stPrcRecipe.stUBL.nRecipeIndexShow.diValue															:=		stPrcRecipe.stUBL.nRecipeIndexShow.diDefault															 ;
stPrcRecipe.stUBL.iPackageCapTypeShow.diValue														:=      stPrcRecipe.stUBL.iPackageCapTypeShow.diDefault														     ;
stPrcRecipe.stUBL.iPackageCapDiameterShow.diValue 													:=      stPrcRecipe.stUBL.iPackageCapDiameterShow.diDefault 													 ;
stPrcRecipe.stUBL.bExEnableShow.bValue 																:=      stPrcRecipe.stUBL.bExEnableShow.bDefault															     ;
stPrcRecipe.stUBL.bBottleFeederEnableShow.bValue													:=      stPrcRecipe.stUBL.bBottleFeederEnableShow.bDefault													     ;
stPrcRecipe.stUBL.iBottleFeederTurntableVelocitySVShow.udiValue										:=      stPrcRecipe.stUBL.iBottleFeederTurntableVelocitySVShow.udiDefault										 ;
stPrcRecipe.stUBL.iBottleFeederBottleSensorDelayShow.diValue										:=      stPrcRecipe.stUBL.iBottleFeederBottleSensorDelayShow.diDefault										     ;
stPrcRecipe.stUBL.iBottleFeederFormGateDelayShow.diValue											:=      stPrcRecipe.stUBL.iBottleFeederFormGateDelayShow.diDefault											     ;
stPrcRecipe.stUBL.iBottleFeederAllowFormDelayShow.diValue											:=      stPrcRecipe.stUBL.iBottleFeederAllowFormDelayShow.diDefault											     ;
stPrcRecipe.stUBL.bPucksInserterEnableShow.bValue													:=      stPrcRecipe.stUBL.bPucksInserterEnableShow.bDefault												         ;
stPrcRecipe.stUBL.iPucksInserterTurntableVelocitySVShow.udiValue 									:=      stPrcRecipe.stUBL.iPucksInserterTurntableVelocitySVShow.udiDefault									     ;
stPrcRecipe.stUBL.iPucksInserterConveyorVelocitySVShow.udiValue										:=      stPrcRecipe.stUBL.iPucksInserterConveyorVelocitySVShow.udiDefault									     ;
stPrcRecipe.stUBL.iPucksInserterBottleSensorDelayShow.diValue										:=      stPrcRecipe.stUBL.iPucksInserterBottleSensorDelayShow.diDefault										     ;
stPrcRecipe.stUBL.iPucksInserterFormGateDelayShow.diValue 											:=      stPrcRecipe.stUBL.iPucksInserterFormGateDelayShow.diDefault 											 ;
stPrcRecipe.stUBL.iPucksInserterAllowFormDelayShow.diValue 											:=      stPrcRecipe.stUBL.iPucksInserterAllowFormDelayShow.diDefault											 ;
stPrcRecipe.stUBL.lrPucksInserterWheelOffsetShow.lrValue 											:=      stPrcRecipe.stUBL.lrPucksInserterWheelOffsetShow.lrDefault											     ;
stPrcRecipe.stUBL.lrPucksInserterWheelAccelerationShow.lrValue 										:=      stPrcRecipe.stUBL.lrPucksInserterWheelAccelerationShow.lrDefault										 ;
stPrcRecipe.stUBL.lrPucksInserterWheelVelocityShow.lrValue 											:=      stPrcRecipe.stUBL.lrPucksInserterWheelVelocityShow.lrDefault											 ;
stPrcRecipe.stUBL.lrPucksInserterHammerHeightSVShow.lrValue 										:=      stPrcRecipe.stUBL.lrPucksInserterHammerHeightSVShow.lrDefault	 										 ;
stPrcRecipe.stUBL.bGateBeforeDispencersEnableShow.bValue											:=      stPrcRecipe.stUBL.bGateBeforeDispencersEnableShow.bDefault									             ;
stPrcRecipe.stUBL.nGateBeforeDispencersTimeFormInsertingShow.lrValue 								:=      stPrcRecipe.stUBL.nGateBeforeDispencersTimeFormInsertingShow.lrDefault								     ;
stPrcRecipe.stUBL.bGateAfterWeightEnableShow.bValue 												:=      stPrcRecipe.stUBL.bGateAfterWeightEnableShow.bDefault												     ;
stPrcRecipe.stUBL.nGateAfterWeightTimeFormInsertingShow.lrValue 									:=      stPrcRecipe.stUBL.nGateAfterWeightTimeFormInsertingShow.lrDefault									     ;
stPrcRecipe.stUBL.bGateRobotEnableShow.bValue       												:=      stPrcRecipe.stUBL.bGateRobotEnableShow.bDefault    												         ;
stPrcRecipe.stUBL.nGateRobotTimeFormInsertingShow.lrValue											:=      stPrcRecipe.stUBL.nGateRobotTimeFormInsertingShow.lrDefault											     ;
stPrcRecipe.stUBL.bFormsDragingLeftEnableShow.bValue         										:=      stPrcRecipe.stUBL.bFormsDragingLeftEnableShow.bDefault       										     ;
stPrcRecipe.stUBL.lrFormsDragingLeftVelocityShow.lrValue         									:=      stPrcRecipe.stUBL.lrFormsDragingLeftVelocityShow.lrDefault	     									     ;
stPrcRecipe.stUBL.lrFormsDragingLeftAccelerationShow.lrValue 										:=      stPrcRecipe.stUBL.lrFormsDragingLeftAccelerationShow.lrDefault											 ;
stPrcRecipe.stUBL.lrFormsDragingLeftDecelerationShow.lrValue   										:=      stPrcRecipe.stUBL.lrFormsDragingLeftDecelerationShow.lrDefault											 ;
stPrcRecipe.stUBL.bFormsDragingRightEnableShow.bValue 												:=      stPrcRecipe.stUBL.bFormsDragingRightEnableShow.bDefault											         ;
stPrcRecipe.stUBL.lrFormsDragingRightVelocityShow.lrValue 											:=      stPrcRecipe.stUBL.lrFormsDragingRightVelocityShow.lrDefault												 ;
stPrcRecipe.stUBL.lrFormsDragingRightAccelerationShow.lrValue 										:=      stPrcRecipe.stUBL.lrFormsDragingRightAccelerationShow.lrDefault											 ;
stPrcRecipe.stUBL.lrFormsDragingRightDecelerationShow.lrValue 										:=      stPrcRecipe.stUBL.lrFormsDragingRightDecelerationShow.lrDefault											 ;
stPrcRecipe.stUBL.bDosingTwoPhasesShow.bValue 	        											:=      stPrcRecipe.stUBL.bDosingTwoPhasesShow.bDefault	        											     ;
stPrcRecipe.stUBL.lrDispencersLifterReadyPositionShow.lrValue 										:=      stPrcRecipe.stUBL.lrDispencersLifterReadyPositionShow.lrDefault									         ;
stPrcRecipe.stUBL.uiDispencerStartDosingDelayShow.udiValue 											:=      stPrcRecipe.stUBL.uiDispencerStartDosingDelayShow.udiDefault									         ;
stPrcRecipe.stUBL.bDispencer1EnableShow.bValue 	          											:=      stPrcRecipe.stUBL.bDispencer1EnableShow.bDefault         											     ;
stPrcRecipe.stUBL.bDispencer2EnableShow.bValue 		  												:=      stPrcRecipe.stUBL.bDispencer2EnableShow.bDefault  												         ;
stPrcRecipe.stUBL.bDispencer3EnableShow.bValue           											:=      stPrcRecipe.stUBL.bDispencer3EnableShow.bDefault        											     ;
stPrcRecipe.stUBL.bDispencer4EnableShow.bValue 			       										:=      stPrcRecipe.stUBL.bDispencer4EnableShow.bDefault	       										         ;
stPrcRecipe.stUBL.lrDispencer1DoseVolumeShow.lrValue 				   								:=      stPrcRecipe.stUBL.lrDispencer1DoseVolumeShow.lrDefault				   								     ;
stPrcRecipe.stUBL.lrDispencer1Phase1VolumeShow.lrValue	           									:=      stPrcRecipe.stUBL.lrDispencer1Phase1VolumeShow.lrDefault	       									     ;
stPrcRecipe.stUBL.lrDispencer1Phase2VolumeShow.lrValue 	       										:=      stPrcRecipe.stUBL.lrDispencer1Phase2VolumeShow.lrDefault	      										 ;
stPrcRecipe.stUBL.lrDispencer1Phase1VelocityShow.lrValue 	       									:=      stPrcRecipe.stUBL.lrDispencer1Phase1VelocityShow.lrDefault	 	       									 ;
stPrcRecipe.stUBL.lrDispencer1Phase2VelocityShow.lrValue 											:=      stPrcRecipe.stUBL.lrDispencer1Phase2VelocityShow.lrDefault	 											 ;
stPrcRecipe.stUBL.lrDispencer1Phase3VelocityShow.lrValue 		   									:=      stPrcRecipe.stUBL.lrDispencer1Phase3VelocityShow.lrDefault	 		   									 ;
stPrcRecipe.stUBL.lrDispencer1SuckVelocityShow.lrValue   											:=      stPrcRecipe.stUBL.lrDispencer1SuckVelocityShow.lrDefault	 											 ;
stPrcRecipe.stUBL.lrDispencer1Phase1AccelerationShow.lrValue 										:=      stPrcRecipe.stUBL.lrDispencer1Phase1AccelerationShow .lrDefault											 ;
stPrcRecipe.stUBL.lrDispencer1Phase2AccelerationShow.lrValue 	  									:=      stPrcRecipe.stUBL.lrDispencer1Phase2AccelerationShow .lrDefault		  									 ;
stPrcRecipe.stUBL.lrDispencer1Phase3AccelerationShow.lrValue 	   									:=      stPrcRecipe.stUBL.lrDispencer1Phase3AccelerationShow .lrDefault		   									 ;
stPrcRecipe.stUBL.lrDispencer1SuckAccelerationShow.lrValue  										:=      stPrcRecipe.stUBL.lrDispencer1SuckAccelerationShow	.lrDefault										     ;
stPrcRecipe.stUBL.lrDispencer1Phase1DecelerationShow.lrValue        								:=      stPrcRecipe.stUBL.lrDispencer1Phase1DecelerationShow  .lrDefault	      								 ;
stPrcRecipe.stUBL.lrDispencer1Phase2DecelerationShow.lrValue 										:=      stPrcRecipe.stUBL.lrDispencer1Phase2DecelerationShow .lrDefault											 ;
stPrcRecipe.stUBL.lrDispencer1Phase3DecelerationShow.lrValue 	   									:=      stPrcRecipe.stUBL.lrDispencer1Phase3DecelerationShow .lrDefault		   									 ;
stPrcRecipe.stUBL.udiDispencer1DosingDoneDelayTimeShow.udiValue 									:=      stPrcRecipe.stUBL.udiDispencer1DosingDoneDelayTimeShow.udiDefault								         ;
stPrcRecipe.stUBL.lrDispencer1SuckValveOpenVolumeShow.lrValue 										:=      stPrcRecipe.stUBL.lrDispencer1SuckValveOpenVolumeShow.lrDefault										     ;
stPrcRecipe.stUBL.lrDispencer1SuckValveOpenTimeDelayShow.lrValue 									:=      stPrcRecipe.stUBL.lrDispencer1SuckValveOpenTimeDelayShow.lrDefault									     ;
stPrcRecipe.stUBL.lrDispencer1SuckValveCloseVolumeShow.lrValue 										:=      stPrcRecipe.stUBL.lrDispencer1SuckValveCloseVolumeShow.lrDefault										 ;
stPrcRecipe.stUBL.lrDispencer1SuckValveCloseTimeDelayShow.lrValue 									:=      stPrcRecipe.stUBL.lrDispencer1SuckValveCloseTimeDelayShow.lrDefault										 ;
stPrcRecipe.stUBL.lrDispencer1DoseValveOpenVolumeShow.lrValue    									:=      stPrcRecipe.stUBL.lrDispencer1DoseValveOpenVolumeShow.lrDefault										     ;
stPrcRecipe.stUBL.lrDispencer1DoseValveOpenTimeAccShow.lrValue   									:=      stPrcRecipe.stUBL.lrDispencer1DoseValveOpenTimeAccShow.lrDefault										 ;
stPrcRecipe.stUBL.lrDispencer1DoseValveCloseVolumeShow.lrValue    									:=      stPrcRecipe.stUBL.lrDispencer1DoseValveCloseVolumeShow.lrDefault									     ;
stPrcRecipe.stUBL.lrDispencer1DoseValveCloseTimeDecShow.lrValue 									:=      stPrcRecipe.stUBL.lrDispencer1DoseValveCloseTimeDecShow.lrDefault									     ;
stPrcRecipe.stUBL.lrDispencer1DoseSuckingVolumeShow.lrValue 										:=      stPrcRecipe.stUBL.lrDispencer1DoseSuckingVolumeShow.lrDefault											 ;
stPrcRecipe.stUBL.lrDispencer1DoseSuckingTimeDelayShow.lrValue 										:=      stPrcRecipe.stUBL.lrDispencer1DoseSuckingTimeDelayShow.lrDefault									     ;
stPrcRecipe.stUBL.bDispencer1DoseSuckingShow.bValue 			       								:=      stPrcRecipe.stUBL.bDispencer1DoseSuckingShow.bDefault	       								             ;
stPrcRecipe.stUBL.bDispencer1LiftSynchroPh1Show.bValue 												:=      stPrcRecipe.stUBL.bDispencer1LiftSynchroPh1Show.bDefault										         ;
stPrcRecipe.stUBL.bDispencer1LiftSynchroPh2Show.bValue 			   									:=      stPrcRecipe.stUBL.bDispencer1LiftSynchroPh2Show.bDefault			   									 ;
stPrcRecipe.stUBL.bDispencer1LiftSynchroPh3Show.bValue 		       									:=      stPrcRecipe.stUBL.bDispencer1LiftSynchroPh3Show.bDefault	       									     ;
stPrcRecipe.stUBL.lrDispencer1LifterStartDosePositionShow.lrValue									:=      stPrcRecipe.stUBL.lrDispencer1LifterStartDosePositionShow.lrDefault									     ;
stPrcRecipe.stUBL.lrDispencer1LifterStopDosePositionShow.lrValue 									:=      stPrcRecipe.stUBL.lrDispencer1LifterStopDosePositionShow.lrDefault										 ;
stPrcRecipe.stUBL.lrDispencer1LifterVelocityShow.lrValue            								:=      stPrcRecipe.stUBL.lrDispencer1LifterVelocityShow.lrDefault	         								     ;
stPrcRecipe.stUBL.lrDispencer1LifterAccelerationShow.lrValue        								:=      stPrcRecipe.stUBL.lrDispencer1LifterAccelerationShow.lrDefault	       								     ;
stPrcRecipe.stUBL.lrDispencer1LifterDecelerationShow.lrValue 		    							:=      stPrcRecipe.stUBL.lrDispencer1LifterDecelerationShow.lrDefault			    							 ;
stPrcRecipe.stUBL.lrDispencer2DoseVolumeShow.lrValue	            								:=      stPrcRecipe.stUBL.lrDispencer2DoseVolumeShow.lrDefault		            								 ;
stPrcRecipe.stUBL.lrDispencer2Phase1VolumeShow.lrValue 			    								:=      stPrcRecipe.stUBL.lrDispencer2Phase1VolumeShow.lrDefault				    							 ;
stPrcRecipe.stUBL.lrDispencer2Phase2VolumeShow.lrValue 			    								:=      stPrcRecipe.stUBL.lrDispencer2Phase2VolumeShow.lrDefault			    								 ;
stPrcRecipe.stUBL.lrDispencer2Phase1VelocityShow.lrValue 		    								:=      stPrcRecipe.stUBL.lrDispencer2Phase1VelocityShow	.lrDefault		    								 ;
stPrcRecipe.stUBL.lrDispencer2Phase2VelocityShow.lrvalue 		    								:=      stPrcRecipe.stUBL.lrDispencer2Phase2VelocityShow	.lrDefault		    								 ;
stPrcRecipe.stUBL.lrDispencer2Phase3VelocityShow.lrValue 		    								:=      stPrcRecipe.stUBL.lrDispencer2Phase3VelocityShow	.lrDefault		    								 ;
stPrcRecipe.stUBL.lrDispencer2SuckVelocityShow.lrValue     											:=      stPrcRecipe.stUBL.lrDispencer2SuckVelocityShow.lrDefault	     										 ;
stPrcRecipe.stUBL.lrDispencer2Phase1AccelerationShow.lrValue 	        							:=      stPrcRecipe.stUBL.lrDispencer2Phase1AccelerationShow.lrDefault		        							 ;
stPrcRecipe.stUBL.lrDispencer2Phase2AccelerationShow.lrValue 	        							:=      stPrcRecipe.stUBL.lrDispencer2Phase2AccelerationShow.lrDefault		        							 ;
stPrcRecipe.stUBL.lrDispencer2Phase3AccelerationShow.lrValue 		    							:=      stPrcRecipe.stUBL.lrDispencer2Phase3AccelerationShow.lrDefault			    							 ;
stPrcRecipe.stUBL.lrDispencer2SuckAccelerationShow.lrValue   										:=      stPrcRecipe.stUBL.lrDispencer2SuckAccelerationShow  .lrDefault	  										 ;
stPrcRecipe.stUBL.lrDispencer2Phase1DecelerationShow.lrValue 										:=      stPrcRecipe.stUBL.lrDispencer2Phase1DecelerationShow.lrDefault											 ;
stPrcRecipe.stUBL.lrDispencer2Phase2DecelerationShow.lrValue 										:=      stPrcRecipe.stUBL.lrDispencer2Phase2DecelerationShow.lrDefault											 ;
stPrcRecipe.stUBL.lrDispencer2Phase3DecelerationShow.lrValue 										:=      stPrcRecipe.stUBL.lrDispencer2Phase3DecelerationShow.lrDefault											 ;
stPrcRecipe.stUBL.udiDispencer2DosingDoneDelayTimeShow.udiValue 									:=      stPrcRecipe.stUBL.udiDispencer2DosingDoneDelayTimeShow.udiDefault								         ;
stPrcRecipe.stUBL.lrDispencer2SuckValveOpenVolumeShow.lrValue 										:=      stPrcRecipe.stUBL.lrDispencer2SuckValveOpenVolumeShow.lrDefault											 ;
stPrcRecipe.stUBL.lrDispencer2SuckValveOpenTimeDelayShow.lrValue 									:=      stPrcRecipe.stUBL.lrDispencer2SuckValveOpenTimeDelayShow.lrDefault										 ;
stPrcRecipe.stUBL.lrDispencer2SuckValveCloseVolumeShow.lrValue										:=      stPrcRecipe.stUBL.lrDispencer2SuckValveCloseVolumeShow.lrDefault										 ;
stPrcRecipe.stUBL.lrDispencer2SuckValveCloseTimeDelayShow.lrValue 									:=      stPrcRecipe.stUBL.lrDispencer2SuckValveCloseTimeDelayShow.lrDefault									     ;
stPrcRecipe.stUBL.lrDispencer2DoseValveOpenVolumeShow.lrValue 										:=      stPrcRecipe.stUBL.lrDispencer2DoseValveOpenVolumeShow .lrDefault										 ;
stPrcRecipe.stUBL.lrDispencer2DoseValveOpenTimeAccShow.lrValue 										:=      stPrcRecipe.stUBL.lrDispencer2DoseValveOpenTimeAccShow.lrDefault										 ; 
stPrcRecipe.stUBL.lrDispencer2DoseValveCloseVolumeShow.lrValue 										:=      stPrcRecipe.stUBL.lrDispencer2DoseValveCloseVolumeShow.lrDefault										 ;
stPrcRecipe.stUBL.lrDispencer2DoseValveCloseTimeDecShow.lrValue										:=      stPrcRecipe.stUBL.lrDispencer2DoseValveCloseTimeDecShow.lrDefault										 ;
stPrcRecipe.stUBL.lrDispencer2DoseSuckingVolumeShow.lrValue	    									:=      stPrcRecipe.stUBL.lrDispencer2DoseSuckingVolumeShow.lrDefault	   									     ;
stPrcRecipe.stUBL.lrDispencer2DoseSuckingTimeDelayShow.lrValue										:=      stPrcRecipe.stUBL.lrDispencer2DoseSuckingTimeDelayShow.lrDefault										 ;
stPrcRecipe.stUBL.bDispencer2DoseSuckingShow.bValue 	            								:=      stPrcRecipe.stUBL.bDispencer2DoseSuckingShow.bDefault            								         ;
stPrcRecipe.stUBL.bDispencer2LiftSynchroPh1Show.bValue 	        									:=      stPrcRecipe.stUBL.bDispencer2LiftSynchroPh1Show.bDefault        									     ;
stPrcRecipe.stUBL.bDispencer2LiftSynchroPh2Show.bValue 	        									:=      stPrcRecipe.stUBL.bDispencer2LiftSynchroPh2Show.bDefault    									         ;
stPrcRecipe.stUBL.bDispencer2LiftSynchroPh3Show.bValue 	        									:=      stPrcRecipe.stUBL.bDispencer2LiftSynchroPh3Show.bDefault 									             ;
stPrcRecipe.stUBL.lrDispencer2LifterStartDosePositionShow.lrValue									:=      stPrcRecipe.stUBL.lrDispencer2LifterStartDosePositionShow.lrDefault									     ;
stPrcRecipe.stUBL.lrDispencer2LifterStopDosePositionShow.lrValue 									:=      stPrcRecipe.stUBL.lrDispencer2LifterStopDosePositionShow .lrDefault								         ;
stPrcRecipe.stUBL.lrDispencer2LifterVelocityShow.lrValue        									:=      stPrcRecipe.stUBL.lrDispencer2LifterVelocityShow.lrDefault	     									     ;
stPrcRecipe.stUBL.lrDispencer2LifterAccelerationShow.lrValue 										:=      stPrcRecipe.stUBL.lrDispencer2LifterAccelerationShow.lrDefault										     ;
stPrcRecipe.stUBL.lrDispencer2LifterDecelerationShow.lrValue 	    								:=      stPrcRecipe.stUBL.lrDispencer2LifterDecelerationShow.lrDefault		    								 ;
stPrcRecipe.stUBL.bDispencersCatchEnableShow.bValue             									:=      stPrcRecipe.stUBL.bDispencersCatchEnableShow.bDefault      									             ;
stPrcRecipe.stUBL.bDispencersCatchMaxPressureShow.bValue          									:=      stPrcRecipe.stUBL.bDispencersCatchMaxPressureShow.bDefault       									     ;
stPrcRecipe.stUBL.lrDispencersCatchHeightSVShow.lrValue												:=      stPrcRecipe.stUBL.lrDispencersCatchHeightSVShow    	.lrDefault									         ;
stPrcRecipe.stUBL.lrDispencersCatch1ClosedValueShow.lrValue          								:=      stPrcRecipe.stUBL.lrDispencersCatch1ClosedValueShow .lrDefault	   								         ;
stPrcRecipe.stUBL.lrDispencersCatch1OpenValueShow.lrValue          									:=      stPrcRecipe.stUBL.lrDispencersCatch1OpenValueShow	 .lrDefault	    									 ;
stPrcRecipe.stUBL.lrDispencersCatch2ClosedValueShow.lrValue       									:=      stPrcRecipe.stUBL.lrDispencersCatch2ClosedValueShow .lrDefault										     ;
stPrcRecipe.stUBL.lrDispencersCatch2OpenValueShow.lrValue	    									:=      stPrcRecipe.stUBL.lrDispencersCatch2OpenValueShow	 .lrDefault	  									     ;
stPrcRecipe.stUBL.lrDispencersCatch3ClosedValueShow.lrValue         								:=      stPrcRecipe.stUBL.lrDispencersCatch3ClosedValueShow  .lrDefault	 								         ;
stPrcRecipe.stUBL.lrDispencersCatch3OpenValueShow.lrValue           								:=      stPrcRecipe.stUBL.lrDispencersCatch3OpenValueShow	  .lrDefault	        							 ;
stPrcRecipe.stUBL.lrDispencersCatch4ClosedValueShow.lrValue         								:=      stPrcRecipe.stUBL.lrDispencersCatch4ClosedValueShow   .lrDefault	 								     ;
stPrcRecipe.stUBL.lrDispencersCatch4OpenValueShow.lrValue											:=      stPrcRecipe.stUBL.lrDispencersCatch4OpenValueShow	.lrDefault										     ;
stPrcRecipe.stUBL.lrDispencersCatchToleranceShow.lrValue 	        								:=      stPrcRecipe.stUBL.lrDispencersCatchToleranceShow	 .lrDefault	      								     ;
stPrcRecipe.stUBL.bTank1MixerEnableShow.bValue    													:=      stPrcRecipe.stUBL.bTank1MixerEnableShow.bDefault													     ;
stPrcRecipe.stUBL.bTankHeatingEnableShow.bValue   													:=      stPrcRecipe.stUBL.bTankHeatingEnableShow.bDefault 													     ;
stPrcRecipe.stUBL.iTankHeatingTempSVShow.diValue  													:=      stPrcRecipe.stUBL.iTankHeatingTempSVShow.diDefault  													 ;
stPrcRecipe.stUBL.bTank1PressureEnableShow.bValue													:=      stPrcRecipe.stUBL.bTank1PressureEnableShow.bDefault											             ;
stPrcRecipe.stUBL.bTank1SupplyPumpEnableShow.bValue                             					:=      stPrcRecipe.stUBL.bTank1SupplyPumpEnableShow.bDefault                        					         ;
stPrcRecipe.stUBL.bTank2SupplyPumpEnableShow.bValue                             					:=      stPrcRecipe.stUBL.bTank2SupplyPumpEnableShow.bDefault                           					     ;
stPrcRecipe.stUBL.uTank1LevelSetpointShow.udiValue                              					:=      stPrcRecipe.stUBL.uTank1LevelSetpointShow.udiDefault                            					     ;
stPrcRecipe.stUBL.uTank2LevelSetpointShow.udiValue                              					:=      stPrcRecipe.stUBL.uTank2LevelSetpointShow.udiDefault                             					     ;
stPrcRecipe.stUBL.bTank1LevelSignalInvertShow.bValue 	                        					:=      stPrcRecipe.stUBL.bTank1LevelSignalInvertShow.bDefault                       					         ;
stPrcRecipe.stUBL.bTank2LevelSignalInvertShow.bValue 	                        					:=      stPrcRecipe.stUBL.bTank2LevelSignalInvertShow.bDefault                        					         ;
stPrcRecipe.stUBL.bWeight1EnableShow.bValue                                     					:=      stPrcRecipe.stUBL.bWeight1EnableShow.bDefault                                   					     ;
stPrcRecipe.stUBL.lrWeightMassSVShow.lrValue	                                					:=      stPrcRecipe.stUBL.lrWeightMassSVShow.lrDefault	                               					         ;
stPrcRecipe.stUBL.iWeight1ActuatorUpDelayShow.diValue 												:=      stPrcRecipe.stUBL.iWeight1ActuatorUpDelayShow.diDefault 												 ;
stPrcRecipe.stUBL.iWeight2ActuatorUpDelayShow.diValue                           					:=      stPrcRecipe.stUBL.iWeight2ActuatorUpDelayShow.diDefault                           					     ;
stPrcRecipe.stUBL.iWeight3ActuatorUpDelayShow.diValue                           					:=      stPrcRecipe.stUBL.iWeight3ActuatorUpDelayShow.diDefault                           					     ;
stPrcRecipe.stUBL.iWeight4ActuatorUpDelayShow.diValue                           					:=      stPrcRecipe.stUBL.iWeight4ActuatorUpDelayShow.diDefault                           					     ;
stPrcRecipe.stUBL.iWeight5ActuatorUpDelayShow.diValue                           					:=      stPrcRecipe.stUBL.iWeight5ActuatorUpDelayShow.diDefault                           					     ;
stPrcRecipe.stUBL.iWeight6ActuatorUpDelayShow.diValue                           					:=      stPrcRecipe.stUBL.iWeight6ActuatorUpDelayShow.diDefault                           					     ;
stPrcRecipe.stUBL.lrFormWeightShow.lrValue                                      					:=      stPrcRecipe.stUBL.lrFormWeightShow	 .lrDefault	                                    					 ;
stPrcRecipe.stUBL.lrMass1DensityShow.lrValue                                    					:=      stPrcRecipe.stUBL.lrMass1DensityShow .lrDefault	                                  					     ;
stPrcRecipe.stUBL.lrMass2DensityShow.lrValue                                    					:=      stPrcRecipe.stUBL.lrMass2DensityShow .lrDefault	                                  					     ;
stPrcRecipe.stUBL.lrCupWeightShow.lrValue                                       					:=      stPrcRecipe.stUBL.lrCupWeightShow	  .lrDefault	                                    				 ;
stPrcRecipe.stUBL.lrWholePackageWeightShow.lrValue 	                            					:=      stPrcRecipe.stUBL.lrWholePackageWeightShow.lrDefault	                           					     ;
stPrcRecipe.stUBL.lrWeight1MeasurmentCorrectionShow.lrValue	                    					:=      stPrcRecipe.stUBL.lrWeight1MeasurmentCorrectionShow.lrDefault	              					         ;
stPrcRecipe.stUBL.bDispencer1WeightCorrectionEnableShow.bValue                  					:=      stPrcRecipe.stUBL.bDispencer1WeightCorrectionEnableShow.bDefault                  					     ;
stPrcRecipe.stUBL.bDispencer2WeightCorrectionEnableShow.bValue                  					:=      stPrcRecipe.stUBL.bDispencer2WeightCorrectionEnableShow.bDefault                  					     ;
stPrcRecipe.stUBL.bDispencer3WeightCorrectionEnableShow.bValue                  					:=      stPrcRecipe.stUBL.bDispencer3WeightCorrectionEnableShow.bDefault                  					     ;
stPrcRecipe.stUBL.bDispencer4WeightCorrectionEnableShow.bValue                  					:=      stPrcRecipe.stUBL.bDispencer4WeightCorrectionEnableShow.bDefault                  					     ;
stPrcRecipe.stUBL.lrWeightUpperToleranceShow.lrValue                            					:=      stPrcRecipe.stUBL.lrWeightUpperToleranceShow.lrDefault	                          					     ;
stPrcRecipe.stUBL.lrWeightLowerToleranceShow.lrValue                            					:=      stPrcRecipe.stUBL.lrWeightLowerToleranceShow.lrDefault	                       					         ;
stPrcRecipe.stUBL.iWeightCorrectionNumberOfSamplesShow.udiValue                 					:=      stPrcRecipe.stUBL.iWeightCorrectionNumberOfSamplesShow.udiDefault            					         ;
stPrcRecipe.stUBL.bLidFeederEnableShow.bValue                 										:=      stPrcRecipe.stUBL.bLidFeederEnableShow.bDefault               										     ;
stPrcRecipe.stUBL.bLidFeederHeaterEnableShow.bValue                             					:=      stPrcRecipe.stUBL.bLidFeederHeaterEnableShow.bDefault                           					     ;
stPrcRecipe.stUBL.lrLidFeederHeightPosSVShow.lrValue                            					:=      stPrcRecipe.stUBL.lrLidFeederHeightPosSVShow.lrDefault	                        					     ;
stPrcRecipe.stUBL.iLidFeederHeatingTimeShow.diValue                             					:=      stPrcRecipe.stUBL.iLidFeederHeatingTimeShow.diDefault                             					     ;
stPrcRecipe.stUBL.iLidFeederTempHisteresisShow.diValue                          					:=      stPrcRecipe.stUBL.iLidFeederTempHisteresisShow.diDefault                          					     ;
stPrcRecipe.stUBL.iLidFeeder1TempSVShow.diValue 	                            					:=      stPrcRecipe.stUBL.iLidFeeder1TempSVShow.diDefault	                            					     ;
stPrcRecipe.stUBL.iLidFeeder2TempSVShow.diValue 	                            					:=      stPrcRecipe.stUBL.iLidFeeder2TempSVShow.diDefault	                            					     ;
stPrcRecipe.stUBL.bLidFeederDragingStationEnableShow.bValue 	                					:=      stPrcRecipe.stUBL.bLidFeederDragingStationEnableShow.bDefault	                					     ;
stPrcRecipe.stUBL.lrLidFeederDragingStationVelocityShow.lrValue	                					:=      stPrcRecipe.stUBL.lrLidFeederDragingStationVelocityShow		.lrDefault		                			 ;	
stPrcRecipe.stUBL.lrLidFeederDragingStationAccelerationShow.lrValue	            					:=      stPrcRecipe.stUBL.lrLidFeederDragingStationAccelerationShow.lrDefault	   					             ;
stPrcRecipe.stUBL.lrLidFeederDragingStationDecelerationShow.lrValue	            					:=      stPrcRecipe.stUBL.lrLidFeederDragingStationDecelerationShow.lrDefault	        					     ;
stPrcRecipe.stUBL.bLidPuttedCheckEnableShow.bValue                              					:=      stPrcRecipe.stUBL.bLidPuttedCheckEnableShow.bDefault                    					             ;
stPrcRecipe.stUBL.lrLidPuttedCheckHeightSVShow.lrValue                          					:=      stPrcRecipe.stUBL.lrLidPuttedCheckHeightSVShow.lrDefault	                   					         ;
stPrcRecipe.stUBL.lrLidPuttedCheckPositionShow.lrValue                          					:=      stPrcRecipe.stUBL.lrLidPuttedCheckPositionShow.lrDefault	                      					     ;
stPrcRecipe.stUBL.lrLidPuttedCheckAreaShow.lrValue                              					:=      stPrcRecipe.stUBL.lrLidPuttedCheckAreaShow.lrDefault	                        					     ;
stPrcRecipe.stUBL.iLidPuttedCheckProgramShow.diValue                            					:=      stPrcRecipe.stUBL.iLidPuttedCheckProgramShow.diDefault                        					         ;
stPrcRecipe.stUBL.bLidSealerEnableShow.bValue                                   					:=      stPrcRecipe.stUBL.bLidSealerEnableShow.bDefault                               					         ;
stPrcRecipe.stUBL.bLidSealerHeaterEnableShow.bValue 	                        					:=      stPrcRecipe.stUBL.bLidSealerHeaterEnableShow.bDefault	                        					     ;
stPrcRecipe.stUBL.iLidSealerHeatingTimeShow.diValue	                            					:=      stPrcRecipe.stUBL.iLidSealerHeatingTimeShow.diDefault                     					             ;
stPrcRecipe.stUBL.lrLidSealerPressureShow.lrValue                               					:=      stPrcRecipe.stUBL.lrLidSealerPressureShow.lrDefault	                           					         ;
stPrcRecipe.stUBL.lrLidSealerHeightPosSVShow.lrValue                            					:=      stPrcRecipe.stUBL.lrLidSealerHeightPosSVShow.lrDefault	                          					     ;
stPrcRecipe.stUBL.iLidSealerTempHisteresisShow.diValue                          					:=      stPrcRecipe.stUBL.iLidSealerTempHisteresisShow.diDefault                    					         ;
stPrcRecipe.stUBL.iLidSealer1TempSVShow.diValue 	                            					:=      stPrcRecipe.stUBL.iLidSealer1TempSVShow.diDefault                            					         ;
stPrcRecipe.stUBL.iLidSealer2TempSVShow.diValue 	                            					:=      stPrcRecipe.stUBL.iLidSealer2TempSVShow.diDefault	                            					     ;
stPrcRecipe.stUBL.bLidSealerDragingStationEnableShow.bValue                     					:=      stPrcRecipe.stUBL.bLidSealerDragingStationEnableShow.bDefault                    					     ;
stPrcRecipe.stUBL.lrLidSealerDragingStationVelocityShow.lrValue 	            					:=      stPrcRecipe.stUBL.lrLidSealerDragingStationVelocityShow.lrDefault	            					     ;
stPrcRecipe.stUBL.lrLidSealerDragingStationAccelerationShow.lrValue	            					:=      stPrcRecipe.stUBL.lrLidSealerDragingStationAccelerationShow.lrDefault	           					     ;
stPrcRecipe.stUBL.lrLidSealerDragingStationDecelerationShow.lrValue	            					:=      stPrcRecipe.stUBL.lrLidSealerDragingStationDecelerationShow.lrDefault	          					     ;
stPrcRecipe.stUBL.bCapFeederGateEnableShow.bValue 	                            					:=      stPrcRecipe.stUBL.bCapFeederGateEnableShow.bDefault	                            					     ;
stPrcRecipe.stUBL.iCapFeederGateBlockingTimeShow.diValue 	                    					:=      stPrcRecipe.stUBL.iCapFeederGateBlockingTimeShow.diDefault	                    					     ;
stPrcRecipe.stUBL.bCapFeederEnableShow.bValue                                   					:=      stPrcRecipe.stUBL.bCapFeederEnableShow.bDefault                              					         ;
stPrcRecipe.stUBL.lrCapFeederHeightPosSVShow.lrValue                            					:=      stPrcRecipe.stUBL.lrCapFeederHeightPosSVShow.lrDefault	                        					     ;
stPrcRecipe.stUBL.iCapFeederTimeDelayOnShow.diValue                             					:=      stPrcRecipe.stUBL.iCapFeederTimeDelayOnShow.diDefault                    					             ;
stPrcRecipe.stUBL.iCapFeederTimeDelayOffShow.diValue                            					:=      stPrcRecipe.stUBL.iCapFeederTimeDelayOffShow.diDefault                     					             ;
stPrcRecipe.stUBL.iCapFeederTimeToEmptySleeveErrorShow.diValue                  					:=      stPrcRecipe.stUBL.iCapFeederTimeToEmptySleeveErrorShow.diDefault             					         ;
stPrcRecipe.stUBL.bCapSorterOnlyWeightOKEnableShow.bValue                       					:=      stPrcRecipe.stUBL.bCapSorterOnlyWeightOKEnableShow.bDefault                 					         ;
stPrcRecipe.stUBL.bCapSorterDragEnableShow.bValue                               					:=      stPrcRecipe.stUBL.bCapSorterDragEnableShow.bDefault                              					     ;
stPrcRecipe.stUBL.lrCapSorterDragVelocityShow.lrValue                           					:=      stPrcRecipe.stUBL.lrCapSorterDragVelocityShow	.lrDefault	                         					 ;
stPrcRecipe.stUBL.lrCapSorterDragAccelerationShow.lrValue 	                    					:=      stPrcRecipe.stUBL.lrCapSorterDragAccelerationShow.lrDefault	                    					     ;
stPrcRecipe.stUBL.lrCapSorterDragDecelerationShow.lrValue 	                    					:=      stPrcRecipe.stUBL.lrCapSorterDragDecelerationShow.lrDefault	               					             ;
stPrcRecipe.stUBL.bCapPuttedCheckEnableShow.bValue                              					:=      stPrcRecipe.stUBL.bCapPuttedCheckEnableShow.bDefault                        					         ;
stPrcRecipe.stUBL.lrCapPuttedCheckHeightPosSVShow.lrValue 	                    					:=      stPrcRecipe.stUBL.lrCapPuttedCheckHeightPosSVShow.lrDefault		                    					 ;
stPrcRecipe.stUBL.bGripperScrewer1EnableShow.bValue 	                        					:=      stPrcRecipe.stUBL.bGripperScrewer1EnableShow.bDefault 	                        					     ;
stPrcRecipe.stUBL.lrGripperScrewingTightTorqueShow.lrValue                      					:=      stPrcRecipe.stUBL.lrGripperScrewingTightTorqueShow.lrDefault	                   					     ;
stPrcRecipe.stUBL.bGripperScrewer2EnableShow.bValue 	                        					:=      stPrcRecipe.stUBL.bGripperScrewer2EnableShow.bDefault	                        					     ;
stPrcRecipe.stUBL.lrGripperScrewing2TightTorqueShow.lrValue	                    					:=      stPrcRecipe.stUBL.lrGripperScrewing2TightTorqueShow.lrDefault	               					         ;
stPrcRecipe.stUBL.iGripperScrewer1ToolShow.diValue                              					:=      stPrcRecipe.stUBL.iGripperScrewer1ToolShow.diDefault                        					         ;
stPrcRecipe.stUBL.lrGripperScrewer1VelocityShow.lrValue                         					:=      stPrcRecipe.stUBL.lrGripperScrewer1VelocityShow.lrDefault	                  					         ;
stPrcRecipe.stUBL.nGripperScrewer1TightTimeShow.diValue	                        					:=      stPrcRecipe.stUBL.nGripperScrewer1TightTimeShow.diDefault                      					         ;
stPrcRecipe.stUBL.iGripperScrewer1StartDelayShow.diValue	                    					:=      stPrcRecipe.stUBL.iGripperScrewer1StartDelayShow.diDefault                    					         ;
stPrcRecipe.stUBL.lrGripperScrewerReadyPositionShow.lrValue 	                					:=      stPrcRecipe.stUBL.lrGripperScrewerReadyPositionShow.lrDefault	                					     ;
stPrcRecipe.stUBL.lrGripperScrewerPushingCapPositionShow.lrValue 	            					:=      stPrcRecipe.stUBL.lrGripperScrewerPushingCapPositionShow.lrDefault	          					         ;
stPrcRecipe.stUBL.lrGripperScrewerScrewingCapPositionShow.lrValue               					:=      stPrcRecipe.stUBL.lrGripperScrewerScrewingCapPositionShow.lrDefault	         					         ;
stPrcRecipe.stUBL.lrGripperScrewerPressureShow.lrValue                          					:=      stPrcRecipe.stUBL.lrGripperScrewerPressureShow.lrDefault	                  					         ;
stPrcRecipe.stUBL.lrGripperScrewerCatchPressureShow.lrValue 	                					:=      stPrcRecipe.stUBL.lrGripperScrewerCatchPressureShow.lrDefault		                					 ;
stPrcRecipe.stUBL.lrDispencerCatchPressureShow.lrValue                          					:=      stPrcRecipe.stUBL.lrDispencerCatchPressureShow.lrDefault	                   					         ;
stPrcRecipe.stUBL.lrGripperScrewerPressureExhaustLevelShow.lrValue              					:=      stPrcRecipe.stUBL.lrGripperScrewerPressureExhaustLevelShow.lrDefault	         					     ;
stPrcRecipe.stUBL.lrGripperScrewerCatchPressureExhaustLevelShow.lrValue         					:=      stPrcRecipe.stUBL.lrGripperScrewerCatchPressureExhaustLevelShow.lrDefault	 					         ;
stPrcRecipe.stUBL.lrGripperScrewerTurnoversToFullScrewedShow.lrValue 	        					:=      stPrcRecipe.stUBL.lrGripperScrewerTurnoversToFullScrewedShow.lrDefault	    					         ;
stPrcRecipe.stUBL.lrGripperScrewerThreadPitchShow.lrValue                       					:=      stPrcRecipe.stUBL.lrGripperScrewerThreadPitchShow.lrDefault	                    					     ;
stPrcRecipe.stUBL.lrGripperScrewerThreadTimesShow.lrValue                       					:=      stPrcRecipe.stUBL.lrGripperScrewerThreadTimesShow.lrDefault	                  					         ;
stPrcRecipe.stUBL.nGripperScrewerCatchHeightSVShow.diValue	                    					:=      stPrcRecipe.stUBL.nGripperScrewerCatchHeightSVShow.diDefault                  					         ;
stPrcRecipe.stUBL.bGripperScrewer1FindScrewShow.bValue                          					:=      stPrcRecipe.stUBL.bGripperScrewer1FindScrewShow.bDefault                					             ;
stPrcRecipe.stUBL.bGripperScrewer1Option4Show.bValue                            					:=      stPrcRecipe.stUBL.bGripperScrewer1Option4Show.bDefault                            					     ;
stPrcRecipe.stUBL.lrGripperScrewer1FindingScrewDegreeShow.lrValue               					:=      stPrcRecipe.stUBL.lrGripperScrewer1FindingScrewDegreeShow.lrDefault	             					     ;
stPrcRecipe.stUBL.bGripperScrewer1Option1Show.bValue	                        					:=      stPrcRecipe.stUBL.bGripperScrewer1Option1Show.bDefault                        					         ;
stPrcRecipe.stUBL.bGripperScrewer1Option2Show.bValue	                        					:=      stPrcRecipe.stUBL.bGripperScrewer1Option2Show.bDefault                        					         ;
stPrcRecipe.stUBL.bGripperScrewer1Option3Show.bValue	                        					:=      stPrcRecipe.stUBL.bGripperScrewer1Option3Show.bDefault                       					         ;
stPrcRecipe.stUBL.bGripperScrewer1Option5Show.bValue	                        					:=      stPrcRecipe.stUBL.bGripperScrewer1Option5Show.bDefault                      					         ;
stPrcRecipe.stUBL.bGripperScrewer1Option6Show.bValue	                        					:=      stPrcRecipe.stUBL.bGripperScrewer1Option6Show.bDefault	                        					     ;
stPrcRecipe.stUBL.bGripperScrewer1Option7Show.bValue	                        					:=      stPrcRecipe.stUBL.bGripperScrewer1Option7Show.bDefault                        					         ;
stPrcRecipe.stUBL.bBottleDragingStationEnableShow.bValue 	                    					:=      stPrcRecipe.stUBL.bBottleDragingStationEnableShow.bDefault	                    					     ;
stPrcRecipe.stUBL.lrBottleDragingStationVelocityShow.lrValue                    					:=      stPrcRecipe.stUBL.lrBottleDragingStationVelocityShow.lrDefault	                   					     ;
stPrcRecipe.stUBL.bCapCorrectCheckEnableShow.bValue 	                        					:=      stPrcRecipe.stUBL.bCapCorrectCheckEnableShow.bDefault	                        					     ;
stPrcRecipe.stUBL.lrCapCorrectCheckHeightPosSVShow.lrValue                      					:=      stPrcRecipe.stUBL.lrCapCorrectCheckHeightPosSVShow.lrDefault	                 					     ;
stPrcRecipe.stUBL.bCapCorrectCheckCameraEnableShow.bValue                       					:=      stPrcRecipe.stUBL.bCapCorrectCheckCameraEnableShow.bDefault                      					     ;
stPrcRecipe.stUBL.iCapCorrectCheckCameraProgramShow.diValue 	                					:=      stPrcRecipe.stUBL.iCapCorrectCheckCameraProgramShow.diDefault	                					     ;
stPrcRecipe.stUBL.bBottleTransferEnableShow.bValue			                    					:=      stPrcRecipe.stUBL.bBottleTransferEnableShow.bDefault	                    					         ;
stPrcRecipe.stUBL.nBottleTransferProgramShow.udiValue			                					:=      stPrcRecipe.stUBL.nBottleTransferProgramShow.udiDefault	                					             ;
stPrcRecipe.stUBL.iBottleTransferPickOffsetXShow.diValue                        					:=      stPrcRecipe.stUBL.iBottleTransferPickOffsetXShow.diDefault                    					         ;
stPrcRecipe.stUBL.iBottleTransferPickOffsetYShow.diValue 	                    					:=      stPrcRecipe.stUBL.iBottleTransferPickOffsetYShow.diDefault                  					         ;
stPrcRecipe.stUBL.iBottleTransferPickOffsetZShow.diValue                        					:=      stPrcRecipe.stUBL.iBottleTransferPickOffsetZShow.diDefault                    					         ;
stPrcRecipe.stUBL.iBottleTransferPick2OffsetXShow.diValue                       					:=      stPrcRecipe.stUBL.iBottleTransferPick2OffsetXShow.diDefault                    					         ;
stPrcRecipe.stUBL.iBottleTransferPick2OffsetYShow.diValue 	                    					:=      stPrcRecipe.stUBL.iBottleTransferPick2OffsetYShow.diDefault                  					         ;
stPrcRecipe.stUBL.iBottleTransferPick2OffsetZShow.diValue                       					:=      stPrcRecipe.stUBL.iBottleTransferPick2OffsetZShow.diDefault                   					         ;
stPrcRecipe.stUBL.iBottleTransferPlace1OffsetXShow.diValue 	                    					:=      stPrcRecipe.stUBL.iBottleTransferPlace1OffsetXShow.diDefault               					             ;
stPrcRecipe.stUBL.iBottleTransferPlace1OffsetYShow.diValue 	                    					:=      stPrcRecipe.stUBL.iBottleTransferPlace1OffsetYShow.diDefault                  					         ;
stPrcRecipe.stUBL.iBottleTransferPlace1OffsetZShow.diValue 	                    					:=      stPrcRecipe.stUBL.iBottleTransferPlace1OffsetZShow.diDefault                   					         ;
stPrcRecipe.stUBL.iBottleTransferPlace2OffsetXShow.diValue 	                    					:=      stPrcRecipe.stUBL.iBottleTransferPlace2OffsetXShow.diDefault                  					         ;
stPrcRecipe.stUBL.iBottleTransferPlace2OffsetYShow.diValue 	                    					:=      stPrcRecipe.stUBL.iBottleTransferPlace2OffsetYShow.diDefault                					         ;
stPrcRecipe.stUBL.iBottleTransferPlace2OffsetZShow.diValue 	                    					:=      stPrcRecipe.stUBL.iBottleTransferPlace2OffsetZShow.diDefault                					         ;
stPrcRecipe.stUBL.iBottleTransferSpeedShow.diValue 	                            					:=      stPrcRecipe.stUBL.iBottleTransferSpeedShow.diDefault                 					                 ;
stPrcRecipe.stUBL.bBottleTransferInkJetEnableShow.bValue 	                    					:=      stPrcRecipe.stUBL.bBottleTransferInkJetEnableShow.bDefault                    					         ;
stPrcRecipe.stUBL.bBottleTransferPickOnlyOneShow.bValue                         					:=      stPrcRecipe.stUBL.bBottleTransferPickOnlyOneShow.bDefault                     					         ;
stPrcRecipe.stUBL.bBottleTransferWeightEnableShow.bValue 	                    					:=      stPrcRecipe.stUBL.bBottleTransferWeightEnableShow.bDefault                  					         ;
stPrcRecipe.stUBL.iBottleTransferWeightIntervalShow.diValue	                    					:=      stPrcRecipe.stUBL.iBottleTransferWeightIntervalShow.diDefault             					             ;
stPrcRecipe.stUBL.bBottleTransferRotateEnableShow.bValue 	                    					:=      stPrcRecipe.stUBL.bBottleTransferRotateEnableShow.bDefault	                    					     ;
stPrcRecipe.stUBL.bBadBottleConveyorEnableShow.bValue                           					:=      stPrcRecipe.stUBL.bBadBottleConveyorEnableShow.bDefault                       					         ;
stPrcRecipe.stUBL.nBadBottleConveyorVelocitySVShow.udiValue 	                					:=      stPrcRecipe.stUBL.nBadBottleConveyorVelocitySVShow.udiDefault                					         ;
stPrcRecipe.stUBL.bLabelMachineEnableShow.bValue 	                            					:=      stPrcRecipe.stUBL.bLabelMachineEnableShow.bDefault                            					         ;
stPrcRecipe.stUBL.bExitTurnTable1EnableShow.bValue                              					:=      stPrcRecipe.stUBL.bExitTurnTable1EnableShow.bDefault                         					         ;
stPrcRecipe.stUBL.bExitConveyorEnableShow.bValue                                					:=      stPrcRecipe.stUBL.bExitConveyorEnableShow.bDefault                          					         ;
stPrcRecipe.stUBL.nExitConveyorVelocitySVShow.udiValue 	                        					:=      stPrcRecipe.stUBL.nExitConveyorVelocitySVShow.udiDefault                    					         ;
stPrcRecipe.stUBL.bFormTransportersEnableShow.bValue						    					:=      stPrcRecipe.stUBL.bFormTransportersEnableShow.bDefault					    					         ;
stPrcRecipe.stUBL.nFormTransportersDispencerVelocitySVShow.udiValue	            					:=      stPrcRecipe.stUBL.nFormTransportersDispencerVelocitySVShow.udiDefault         					         ;
stPrcRecipe.stUBL.nFormTransportersScrewerVelocitySVShow.udiValue			    					:=      stPrcRecipe.stUBL.nFormTransportersScrewerVelocitySVShow.udiDefault	    					             ;
stPrcRecipe.stUBL.nFormTransportersBeforeScrewerVelocitySVShow.udiValue	        					:=      stPrcRecipe.stUBL.nFormTransportersBeforeScrewerVelocitySVShow.udiDefault    					         ;
stPrcRecipe.stUBL.nFormTransportersSlowerVelocitySVShow.udiValue		 	    					:=      stPrcRecipe.stUBL.nFormTransportersSlowerVelocitySVShow.udiDefault 	    					             ;
stPrcRecipe.stUBL.bCircularInkjetEnableShow.bValue	 	                        					:=      stPrcRecipe.stUBL.bCircularInkjetEnableShow.bDefault	                        					     ;
stPrcRecipe.stUBL.iCircularInkjetSpeedShow.diValue	 	                        					:=      stPrcRecipe.stUBL.iCircularInkjetSpeedShow.diDefault 	                        					     ;
stPrcRecipe.stUBL.iCircularInkjetDelayShow.diValue	 	                        					:=      stPrcRecipe.stUBL.iCircularInkjetDelayShow.diDefault	                        					     ;
stPrcRecipe.stUBL.iCircularInkjetHoldShow.diValue	 	                        					:=      stPrcRecipe.stUBL.iCircularInkjetHoldShow.diDefault	 	                        					     ;
stPrcRecipe.stUCF.iCapSorterProductType.diValue 	                            					:=      stPrcRecipe.stUCF.iCapSorterProductType.diDefault	                            					     ;
stPrcRecipe.stUCF.uiCapSorterIndexShow.udiValue 													:=      stPrcRecipe.stUCF.uiCapSorterIndexShow.udiDefault												         ;
stPrcRecipe.stUCF.bPresenceBottleEnableShow.bValue 	                            					:=      stPrcRecipe.stUCF.bPresenceBottleEnableShow.bDefault                          					         ;
stPrcRecipe.stUCF.bCapSorterTransporterEnableShow.bValue											:=      stPrcRecipe.stUCF.bCapSorterTransporterEnableShow.bDefault											     ;
stPrcRecipe.stUCF.iCapSorterTransporterTankConveyorVelocityShow.diValue								:=      stPrcRecipe.stUCF.iCapSorterTransporterTankConveyorVelocityShow.diDefault						         ;
stPrcRecipe.stUCF.iCapSorterTransporterStartDelayTimeShow.diValue									:=      stPrcRecipe.stUCF.iCapSorterTransporterStartDelayTimeShow.diDefault							             ;
stPrcRecipe.stUCF.udiCapSorterTransporterTimeProductOnSensorBeforeBrushShow.udiValue				:=      stPrcRecipe.stUCF.udiCapSorterTransporterTimeProductOnSensorBeforeBrushShow.udiDefault			         ;
stPrcRecipe.stUCF.iCapSorterTransporterEmptyingConveyorSpeedShow.diValue							:=      stPrcRecipe.stUCF.iCapSorterTransporterEmptyingConveyorSpeedShow.diDefault							     ;
stPrcRecipe.stUCF.iCapSorterTransporterVolumeOfCapsShow.diValue										:=      stPrcRecipe.stUCF.iCapSorterTransporterVolumeOfCapsShow.diDefault							             ;
stPrcRecipe.stUCF.bCapSorterWheelEnableShow.bValue							    					:=      stPrcRecipe.stUCF.bCapSorterWheelEnableShow.bDefault						    					     ;
stPrcRecipe.stUCF.lrCapSorterWheelMoveAccelerationEmptyTableShow.lrValue	    					:=      stPrcRecipe.stUCF.lrCapSorterWheelMoveAccelerationEmptyTableShow.lrDefault	  					         ;
stPrcRecipe.stUCF.lrCapSorterWheelMoveDecelerationEmptyTableShow.lrValue	    					:=      stPrcRecipe.stUCF.lrCapSorterWheelMoveDecelerationEmptyTableShow.lrDefault	    					     ;
stPrcRecipe.stUCF.lrCapSorterWheelMoveSpeedEmptyTableShow.lrValue			    					:=      stPrcRecipe.stUCF.lrCapSorterWheelMoveSpeedEmptyTableShow.lrDefault			    					     ;
stPrcRecipe.stUCF.lrCapSorterWheelMoveAngleEmptyTableShow.lrValue			    					:=      stPrcRecipe.stUCF.lrCapSorterWheelMoveAngleEmptyTableShow.lrDefault			    					     ;
stPrcRecipe.stUCF.lrCapSorterWheelJerkAngleEmptyTableShow.lrValue			    					:=      stPrcRecipe.stUCF.lrCapSorterWheelJerkAngleEmptyTableShow.lrDefault		    					         ;
stPrcRecipe.stUCF.iCapSorterWheelWaitingAfterRotationEmptyTableShow.diValue     					:=      stPrcRecipe.stUCF.iCapSorterWheelWaitingAfterRotationEmptyTableShow.diDefault 					         ;
stPrcRecipe.stUCF.lrCapSorterWheelMoveAccelerationFullTableShow.lrValue	        					:=      stPrcRecipe.stUCF.lrCapSorterWheelMoveAccelerationFullTableShow.lrDefault	     					     ;
stPrcRecipe.stUCF.lrCapSorterWheelMoveDecelerationFullTableShow.lrValue	        					:=      stPrcRecipe.stUCF.lrCapSorterWheelMoveDecelerationFullTableShow.lrDefault	  					         ;
stPrcRecipe.stUCF.lrCapSorterWheelMoveSpeedFullTableShow.lrValue			    					:=      stPrcRecipe.stUCF.lrCapSorterWheelMoveSpeedFullTableShow.lrDefault		    					         ;
stPrcRecipe.stUCF.lrCapSorterWheelMoveAngleFullyTableShow.lrValue			    					:=      stPrcRecipe.stUCF.lrCapSorterWheelMoveAngleFullyTableShow.lrDefault			    					     ;
stPrcRecipe.stUCF.lrCapSorterWheelJerkAngleFullTableShow.lrValue			    					:=      stPrcRecipe.stUCF.lrCapSorterWheelJerkAngleFullTableShow.lrDefault				    					 ;
stPrcRecipe.stUCF.iCapSorterWheelWaitingAfterRotationFullTableShow.diValue      					:=      stPrcRecipe.stUCF.iCapSorterWheelWaitingAfterRotationFullTableShow.diDefault    					     ;
stPrcRecipe.stUCF.lrCapSorterWheelMoveAccelerationHalfFullTableShow.lrValue     					:=      stPrcRecipe.stUCF.lrCapSorterWheelMoveAccelerationHalfFullTableShow.lrDefault	   					     ;
stPrcRecipe.stUCF.lrCapSorterWheelMoveDecelerationHalfFullTableShow.lrValue     					:=      stPrcRecipe.stUCF.lrCapSorterWheelMoveDecelerationHalfFullTableShow.lrDefault	 					     ;
stPrcRecipe.stUCF.lrCapSorterWheelMoveSpeedHalfFullTableShow.lrValue								:=      stPrcRecipe.stUCF.lrCapSorterWheelMoveSpeedHalfFullTableShow.lrDefault								     ;
stPrcRecipe.stUCF.lrCapSorterWheelMoveAngleHalfFullyTableShow.lrValue								:=      stPrcRecipe.stUCF.lrCapSorterWheelMoveAngleHalfFullyTableShow.lrDefault							         ;
stPrcRecipe.stUCF.lrCapSorterWheelJerkAngleHalfFullTableShow.lrValue								:=      stPrcRecipe.stUCF.lrCapSorterWheelJerkAngleHalfFullTableShow.lrDefault								     ;
stPrcRecipe.stUCF.iCapSorterWheelWaitingAfterRotationHalfFullTableShow.diValue 						:=      stPrcRecipe.stUCF.iCapSorterWheelWaitingAfterRotationHalfFullTableShow.diDefault				         ;
stPrcRecipe.stUCF.bCapSorterCameraEnableShow.bValue                            						:=      stPrcRecipe.stUCF.bCapSorterCameraEnableShow.bDefault                         						     ;
stPrcRecipe.stUCF.bCapSorterRobotEnableShow.bValue                 			    					:=      stPrcRecipe.stUCF.bCapSorterRobotEnableShow.bDefault               			    					     ;
stPrcRecipe.stUCF.lrCapSorterRobotPlace1PositionXShow.lrValue										:=      stPrcRecipe.stUCF.lrCapSorterRobotPlace1PositionXShow.lrDefault										     ;
stPrcRecipe.stUCF.lrCapSorterRobotPlace1PositionYShow.lrValue										:=      stPrcRecipe.stUCF.lrCapSorterRobotPlace1PositionYShow.lrDefault										     ;
stPrcRecipe.stUCF.lrCapSorterRobotPlace1PositionZShow.lrValue										:=      stPrcRecipe.stUCF.lrCapSorterRobotPlace1PositionZShow.lrDefault										     ;
stPrcRecipe.stUCF.lrCapSorterRobotPlace1PositionCShow.lrValue										:=      stPrcRecipe.stUCF.lrCapSorterRobotPlace1PositionCShow.lrDefault										     ;
stPrcRecipe.stUCF.iCapSorterRobotPickElevationShow.diValue											:=      stPrcRecipe.stUCF.iCapSorterRobotPickElevationShow.diDefault										     ;
stPrcRecipe.stUCF.iCapSorterRobotPickTimeShow.diValue												:=      stPrcRecipe.stUCF.iCapSorterRobotPickTimeShow.diDefault										             ;
stPrcRecipe.stUCF.iCapSorterRobotVacuumActivationShow.diValue										:=      stPrcRecipe.stUCF.iCapSorterRobotVacuumActivationShow.diDefault									         ;
stPrcRecipe.stUCF.iCapSorterRobotVacuumOffShow.diValue						    					:=      stPrcRecipe.stUCF.iCapSorterRobotVacuumOffShow.diDefault				    					         ;
stPrcRecipe.stUCF.iCapSorterRobotPlaceTimeShow.diValue												:=      stPrcRecipe.stUCF.iCapSorterRobotPlaceTimeShow.diDefault										         ;
stPrcRecipe.stUCF.iCapSorterRobotTCP_PlaceOffsetShow.diValue			    						:=      stPrcRecipe.stUCF.iCapSorterRobotTCP_PlaceOffsetShow.diDefault		    						         ;
stPrcRecipe.stUCF.iCapSorterRobotAccelerationDecelerationShow.diValue	 							:=      stPrcRecipe.stUCF.iCapSorterRobotAccelerationDecelerationShow.diDefault 							     ;
stPrcRecipe.stUCF.iCapSorterRobotGripperWatchdogShow.diValue			    						:=      stPrcRecipe.stUCF.iCapSorterRobotGripperWatchdogShow.diDefault		    						         ;
stPrcRecipe.stUCF.iCapSorterRobotParalaxCorrectionShow.diValue		    							:=      stPrcRecipe.stUCF.iCapSorterRobotParalaxCorrectionShow.diDefault    							         ;
stPrcRecipe.stUCF.iCapSorterRobotNumberToolShow.diValue		 										:=      stPrcRecipe.stUCF.iCapSorterRobotNumberToolShow.diDefault	 										     ;
stPrcRecipe.stUCF.iCapSorterRobotPickPositionZShow.diValue 											:=      stPrcRecipe.stUCF.iCapSorterRobotPickPositionZShow.diDefault										     ;
stPrcRecipe.stUCF.iCapSorterRobotTCP_Lenght.diValue		 											:=      stPrcRecipe.stUCF.iCapSorterRobotTCP_Lenght.diDefault											         ;
stPrcRecipe.stUCF.iCapSorterRobotProductDiametr.diValue	 											:=      stPrcRecipe.stUCF.iCapSorterRobotProductDiametr.diDefault									             ;
stPrcRecipe.stUCF.bCapSorterIntermediateTransporterEnableShow.bValue								:=      stPrcRecipe.stUCF.bCapSorterIntermediateTransporterEnableShow.bDefault								     ;
stPrcRecipe.stUCF.iCapSorterIntermediateTransporterAutoSpeedShow.diValue							:=      stPrcRecipe.stUCF.iCapSorterIntermediateTransporterAutoSpeedShow.diDefault							     ;
stPrcRecipe.stUCF.iCapSorterIntermediateTransporterManualSpeedShow.diValue							:=      stPrcRecipe.stUCF.iCapSorterIntermediateTransporterManualSpeedShow.diDefault					         ;
stPrcRecipe.stUCF.iCapSorterIntermediateTransporterEmptyingSpeedShow.diValue						:=      stPrcRecipe.stUCF.iCapSorterIntermediateTransporterEmptyingSpeedShow.diDefault			                 ;
stPrcRecipe.stUCF.iCapSorterIntermediateTransporterDelayCountTimeShow.diValue						:=      stPrcRecipe.stUCF.iCapSorterIntermediateTransporterDelayCountTimeShow.diDefault				             ;
stPrcRecipe.stUCF.iCapSorterIntermediateTransporterReverseTimeShow.diValue							:=      stPrcRecipe.stUCF.iCapSorterIntermediateTransporterReverseTimeShow.diDefault						     ;
stPrcRecipe.stUCF.udiCapSorterIntermediateTransporterTimeProductOnSensorShow.udiValue 				:=      stPrcRecipe.stUCF.udiCapSorterIntermediateTransporterTimeProductOnSensorShow.udiDefault	                 ;
stPrcRecipe.stUCF.lrCapSorterIntermediateTransporterWheelAngleShow.lrValue							:=      stPrcRecipe.stUCF.lrCapSorterIntermediateTransporterWheelAngleShow.lrDefault							 ;
stPrcRecipe.stUCF.bCapSorterIntermediateBrushEnableShow.bValue			 	    					:=      stPrcRecipe.stUCF.bCapSorterIntermediateBrushEnableShow.bDefault	 	    					         ;
stPrcRecipe.stUCF.iCapSorterIntermediateBrushAutoSpeedShow.diValue		 	    					:=      stPrcRecipe.stUCF.iCapSorterIntermediateBrushAutoSpeedShow.diDefault	 	    					     ;
stPrcRecipe.stUCF.iCapSorterIntermediateBrushManualSpeedShow.diValue		  						:=      stPrcRecipe.stUCF.iCapSorterIntermediateBrushManualSpeedShow.diDefault		  						     ;
stPrcRecipe.stUCF.iCapSorterIntermediateBrushEmptyingSpeedShow.diValue	 	    					:=      stPrcRecipe.stUCF.iCapSorterIntermediateBrushEmptyingSpeedShow.diDefault	    					     ;
stPrcRecipe.stUCF.lrCapSorterIntermediateBrushPositionHeightSVShow.lrValue 							:=      stPrcRecipe.stUCF.lrCapSorterIntermediateBrushPositionHeightSVShow.lrDefault								;
stPrcRecipe.stUCF.bCapSorterBrush1OnWheelEnableShow.bValue			  								:=      stPrcRecipe.stUCF.bCapSorterBrush1OnWheelEnableShow.bDefault	  								         ;
stPrcRecipe.stUCF.iCapSorterBrush1OnWheelAutoSpeedShow.diValue		  								:=      stPrcRecipe.stUCF.iCapSorterBrush1OnWheelAutoSpeedShow.diDefault	  								     ;
stPrcRecipe.stUCF.iCapSorterBrush1OnWheelManualSpeedShow.diValue		     						:=      stPrcRecipe.stUCF.iCapSorterBrush1OnWheelManualSpeedShow.diDefault		     						     ;
stPrcRecipe.stUCF.iCapSorterBrush1OnWheelEmptyingSpeedShow.diValue	  								:=      stPrcRecipe.stUCF.iCapSorterBrush1OnWheelEmptyingSpeedShow.diDefault  								     ;
stPrcRecipe.stUCF.lrCapSorterBrush1OnWheelPositionHeightSVShow.lrValue   							:=      stPrcRecipe.stUCF.lrCapSorterBrush1OnWheelPositionHeightSVShow.lrDefault							     ;
stPrcRecipe.stUCF.bCapSorterBrush2OnWheelEnableShow.bValue			 								:=      stPrcRecipe.stUCF.bCapSorterBrush2OnWheelEnableShow.bDefault			 								 ;
stPrcRecipe.stUCF.iCapSorterBrush2OnWheelAutoSpeedShow.diValue		 								:=      stPrcRecipe.stUCF.iCapSorterBrush2OnWheelAutoSpeedShow.diDefault 								         ;
stPrcRecipe.stUCF.iCapSorterBrush2OnWheelManualSpeedShow.diValue	      							:=      stPrcRecipe.stUCF.iCapSorterBrush2OnWheelManualSpeedShow.diDefault	      							     ;
stPrcRecipe.stUCF.iCapSorterBrush2OnWheelEmptyingSpeedShow.diValue	   								:=      stPrcRecipe.stUCF.iCapSorterBrush2OnWheelEmptyingSpeedShow.diDefault 								     ;
stPrcRecipe.stUCF.lrCapSorterBrush2OnWheelPositionHeightSVShow.lrValue   							:=      stPrcRecipe.stUCF.lrCapSorterBrush2OnWheelPositionHeightSVShow.lrDefault							     ;
stPrcRecipe.stUCF.bCapSorterFeederEnableShow.bValue													:=      stPrcRecipe.stUCF.bCapSorterFeederEnableShow.bDefault											         ;
stPrcRecipe.stUCF.bCapSorterFeederEnableTubeError.bValue											:=      stPrcRecipe.stUCF.bCapSorterFeederEnableTubeError.bDefault										         ;
stPrcRecipe.stUCF.lrCapSorterFeederMover1InputPositionShow.lrValue									:=      stPrcRecipe.stUCF.lrCapSorterFeederMover1InputPositionShow.lrDefault								     ;
stPrcRecipe.stUCF.lrCapSorterFeederMover2InputPositionShow.lrValue									:=      stPrcRecipe.stUCF.lrCapSorterFeederMover2InputPositionShow.lrDefault								     ;
stPrcRecipe.stUCF.lrCapSorterFeederMover1OutputPositionShow.lrValue									:=      stPrcRecipe.stUCF.lrCapSorterFeederMover1OutputPositionShow.lrDefault								     ;
stPrcRecipe.stUCF.lrCapSorterFeederMover2OutputPositionShow.lrValue									:=      stPrcRecipe.stUCF.lrCapSorterFeederMover2OutputPositionShow.lrDefault								     ;
stPrcRecipe.stUCF.lrCapSorterFeederSlotDistanceShow.lrValue											:=      stPrcRecipe.stUCF.lrCapSorterFeederSlotDistanceShow.lrDefault									         ;
stPrcRecipe.stUCF.lrCapSorterFeederMoverSpeedShow.lrValue											:=      stPrcRecipe.stUCF.lrCapSorterFeederMoverSpeedShow.lrDefault											     ;
stPrcRecipe.stUCF.lrCapSorterFeederMoverAccelerationShow.lrValue    								:=      stPrcRecipe.stUCF.lrCapSorterFeederMoverAccelerationShow.lrDefault								         ;
stPrcRecipe.stUCF.lrCapSorterFeederMoveJerkShow.lrValue												:=      stPrcRecipe.stUCF.lrCapSorterFeederMoveJerkShow.lrDefault											     ;
stPrcRecipe.stUCF.bCapSorterPreScrewerEnableShow.bValue												:=      stPrcRecipe.stUCF.bCapSorterPreScrewerEnableShow.bDefault										         ;
stPrcRecipe.stUCF.bCapSorterPreScrewerPicker1EnableShow.bValue           							:=      stPrcRecipe.stUCF.bCapSorterPreScrewerPicker1EnableShow.bDefault        							     ;
stPrcRecipe.stUCF.bCapSorterPreScrewerPicker2EnableShow.bValue           							:=      stPrcRecipe.stUCF.bCapSorterPreScrewerPicker2EnableShow.bDefault        							     ;
stPrcRecipe.stUCF.bCapSorterPreScrewerPicker3EnableShow.bValue          							:=      stPrcRecipe.stUCF.bCapSorterPreScrewerPicker3EnableShow.bDefault        							     ;
stPrcRecipe.stUCF.bCapSorterPreScrewerPicker4EnableShow.bValue          							:=      stPrcRecipe.stUCF.bCapSorterPreScrewerPicker4EnableShow.bDefault        							     ;
stPrcRecipe.stUCF.lrCapSorterPreScrewerPickZPositionShow.lrValue									:=      stPrcRecipe.stUCF.lrCapSorterPreScrewerPickZPositionShow.lrDefault									     ;
stPrcRecipe.stUCF.lrCapSorterPreScrewerCatcherReleseShow.lrValue									:=      stPrcRecipe.stUCF.lrCapSorterPreScrewerCatcherReleseShow.lrDefault									     ;
stPrcRecipe.stUCF.lrCapSorterPreScrewerCapCatcherZPositionShow.lrValue								:=      stPrcRecipe.stUCF.lrCapSorterPreScrewerCapCatcherZPositionShow.lrDefault								 ;
stPrcRecipe.stUCF.lrCapSorterPreScrewerTopZPositionShow.lrValue										:=      stPrcRecipe.stUCF.lrCapSorterPreScrewerTopZPositionShow.lrDefault									     ;
stPrcRecipe.stUCF.lrCapSorterPreScrewerCartesianCatchZPositionShow.lrValue							:=      stPrcRecipe.stUCF.lrCapSorterPreScrewerCartesianCatchZPositionShow.lrDefault							 ;
stPrcRecipe.stUCF.lrCapSorterPreScrewerStrawCatcherZPositionShow.lrValue							:=      stPrcRecipe.stUCF.lrCapSorterPreScrewerStrawCatcherZPositionShow.lrDefault							     ;
stPrcRecipe.stUCF.LrCapSorterPreScrewerCheckStrawCatcherActuatorZPosition.lrValue 					:=      stPrcRecipe.stUCF.LrCapSorterPreScrewerCheckStrawCatcherActuatorZPosition.lrDefault					     ;
stPrcRecipe.stUCF.lrCapSorterPreScrewerScrewerStartZPositionShow.lrValue							:=      stPrcRecipe.stUCF.lrCapSorterPreScrewerScrewerStartZPositionShow.lrDefault								 ;
stPrcRecipe.stUCF.lrCapSorterPreScrewerGripperOpenPositionShow.lrValue								:=      stPrcRecipe.stUCF.lrCapSorterPreScrewerGripperOpenPositionShow.lrDefault								 ;
stPrcRecipe.stUCF.lrCapSorterPreScrewerPlaceZPositionShow.lrValue									:=      stPrcRecipe.stUCF.lrCapSorterPreScrewerPlaceZPositionShow.lrDefault									     ;
stPrcRecipe.stUCF.lrCapSorterPreScrewerBendingDistanceShow.lrValue              					:=      stPrcRecipe.stUCF.lrCapSorterPreScrewerBendingDistanceShow.lrDefault	          					     ;
stPrcRecipe.stUCF.lrCapSorterPreScrewerStrawInsertDistance.lrValue              					:=      stPrcRecipe.stUCF.lrCapSorterPreScrewerStrawInsertDistance.lrDefault	            					 ;
stPrcRecipe.stUCF.lrCapSorterPreScrewerPickXMover1PositionShow.lrValue          					:=      stPrcRecipe.stUCF.lrCapSorterPreScrewerPickXMover1PositionShow.lrDefault	       					     ;
stPrcRecipe.stUCF.lrCapSorterPreScrewerPickXMover2PositionShow.lrValue          					:=      stPrcRecipe.stUCF.lrCapSorterPreScrewerPickXMover2PositionShow.lrDefault	         					 ;
stPrcRecipe.stUCF.lrCapSorterPreScrewerPlaceXPositionShow.lrValue		        					:=      stPrcRecipe.stUCF.lrCapSorterPreScrewerPlaceXPositionShow.lrDefault		        					     ;
stPrcRecipe.stUCF.lrCapSorterPreScrewerScrewFindingShow.lrValue	                					:=      stPrcRecipe.stUCF.lrCapSorterPreScrewerScrewFindingShow.lrDefault	              					     ;
stPrcRecipe.stUCF.lrCapSorterPreScrewerScrewDistanceShow.lrValue                					:=      stPrcRecipe.stUCF.lrCapSorterPreScrewerScrewDistanceShow.lrDefault	               					     ;
stPrcRecipe.stUCF.lrCapSorterPreScrewerPickerSpeedShow.lrValue		            					:=      stPrcRecipe.stUCF.lrCapSorterPreScrewerPickerSpeedShow.lrDefault		            					 ;
stPrcRecipe.stUCF.lrCapSorterPreScrewerPickerAccelerationShow.lrValue	        					:=      stPrcRecipe.stUCF.lrCapSorterPreScrewerPickerAccelerationShow.lrDefault	      					         ;
stPrcRecipe.stUCF.lrCapSorterPreScrewerPickerJerkShow.lrValue			        					:=      stPrcRecipe.stUCF.lrCapSorterPreScrewerPickerJerkShow.lrDefault			        					     ;
stPrcRecipe.stUCF.lrCapSorterPreScrewerCatcherSpeedShow.lrValue		            					:=      stPrcRecipe.stUCF.lrCapSorterPreScrewerCatcherSpeedShow.lrDefault	            					     ;
stPrcRecipe.stUCF.lrCapSorterPreScrewerCatcherAccelerationShow.lrValue          					:=      stPrcRecipe.stUCF.lrCapSorterPreScrewerCatcherAccelerationShow.lrDefault	        					 ;
stPrcRecipe.stUCF.lrCapSorterPreScrewerCatcherJerkShow.lrValue		            					:=      stPrcRecipe.stUCF.lrCapSorterPreScrewerCatcherJerkShow.lrDefault	            					     ;
stPrcRecipe.stUCF.lrCapSorterPreScrewerScrewSpeedShow.lrValue			        					:=      stPrcRecipe.stUCF.lrCapSorterPreScrewerScrewSpeedShow.lrDefault			        					     ;
stPrcRecipe.stUCF.lrCapSorterPreScrewerScrewAccelerationShow.lrValue	        					:=      stPrcRecipe.stUCF.lrCapSorterPreScrewerScrewAccelerationShow.lrDefault		        					 ;
stPrcRecipe.stUCF.lrCapSorterPreScrewerScrewJerkShow.lrValue			        					:=      stPrcRecipe.stUCF.lrCapSorterPreScrewerScrewJerkShow.lrDefault			        					     ;
stPrcRecipe.stUCF.lrCapSorterPreScrewerCatcherCatchingPositionShow.lrValue      					:=      stPrcRecipe.stUCF.lrCapSorterPreScrewerCatcherCatchingPositionShow.lrDefault						     ;
stPrcRecipe.stUCF.lrCapSorterPreScrewerCatcherPlacePositionShow.lrValue	        					:=      stPrcRecipe.stUCF.lrCapSorterPreScrewerCatcherPlacePositionShow.lrDefault	   					         ;
stPrcRecipe.stUCF.lrCapSorterPreScrewerCatcherHightSVShow.lrValue			    					:=      stPrcRecipe.stUCF.lrCapSorterPreScrewerCatcherHightSVShow.lrDefault			    					     ;
stPrcRecipe.stUCF.bCapSorterPreScrewerBottleCatcherEnableShow.bValue		    					:=      stPrcRecipe.stUCF.bCapSorterPreScrewerBottleCatcherEnableShow.bDefault		    					     ;
stPrcRecipe.stUCF.lrCapSorterPreScrewerBottleCatch1OpenValueShow.lrValue	    					:=      stPrcRecipe.stUCF.lrCapSorterPreScrewerBottleCatch1OpenValueShow.lrDefault		    					 ;
stPrcRecipe.stUCF.lrCapSorterPreScrewerBottleCatch1CloseValueShow.lrValue	    					:=      stPrcRecipe.stUCF.lrCapSorterPreScrewerBottleCatch1CloseValueShow.lrDefault	   					         ;
stPrcRecipe.stUCF.lrCapSorterPreScrewerBottleCatch2OpenValueShow.lrValue	    					:=      stPrcRecipe.stUCF.lrCapSorterPreScrewerBottleCatch2OpenValueShow.lrDefault	    					     ;
stPrcRecipe.stUCF.lrCapSorterPreScrewerBottleCatch2CloseValueShow.lrValue	    					:=      stPrcRecipe.stUCF.lrCapSorterPreScrewerBottleCatch2CloseValueShow.lrDefault	 					         ;
stPrcRecipe.stUCF.lrCapSorterPreScrewerBottleCatch3OpenValueShow.lrValue	    					:=      stPrcRecipe.stUCF.lrCapSorterPreScrewerBottleCatch3OpenValueShow.lrDefault	  					         ;
stPrcRecipe.stUCF.lrCapSorterPreScrewerBottleCatch3CloseValueShow.lrValue	    					:=      stPrcRecipe.stUCF.lrCapSorterPreScrewerBottleCatch3CloseValueShow.lrDefault	  					         ;
stPrcRecipe.stUCF.lrCapSorterPreScrewerBottleCatch4OpenValueShow.lrValue	                      	:=      stPrcRecipe.stUCF.lrCapSorterPreScrewerBottleCatch4OpenValueShow.lrDefault	                     	     ;
stPrcRecipe.stUCF.lrCapSorterPreScrewerBottleCatch4CloseValueShow.lrValue	                      	:=      stPrcRecipe.stUCF.lrCapSorterPreScrewerBottleCatch4CloseValueShow.lrDefault	                  	         ;
stPrcRecipe.stUCF.lrCapSorterPreScrewerBottleCatchToleranceValueShow.lrValue                      	:=      stPrcRecipe.stUCF.lrCapSorterPreScrewerBottleCatchToleranceValueShow.lrDefault	                    	 ;
stPrcRecipe.stUCF.lrCapSorterPreScrewerCatchAngleOpenSV.lrValue                       				:=      stPrcRecipe.stUCF.lrCapSorterPreScrewerCatchAngleOpenSV.lrDefault	                    				 ;
stPrcRecipe.stUCF.lrCapSorterPreScrewerWaitInPlaceTimeShow.lrValue                                	:=      stPrcRecipe.stUCF.lrCapSorterPreScrewerWaitInPlaceTimeShow.lrDefault	                                	;
stPrcRecipe.stUCF.bCapSorterPreScrewerCatchAngleOpenEnaShow.bValue                                	:=      stPrcRecipe.stUCF.bCapSorterPreScrewerCatchAngleOpenEnaShow.bDefault                              	     ;
stPrcRecipe.stUCF.bCapSorterPreScrewerPoundedInCap.bValue                       					:=      stPrcRecipe.stUCF.bCapSorterPreScrewerPoundedInCap.bDefault                  					         ;
stPrcRecipe.stUCF.lrCapSorterBottleHightShow.lrValue		                                      	:=      stPrcRecipe.stUCF.lrCapSorterBottleHightShow.lrDefault		                                      	     ;
stPrcRecipe.stUCF.lrCapSorterBottleNeckHightShow.lrValue	                                      	:=      stPrcRecipe.stUCF.lrCapSorterBottleNeckHightShow.lrDefault	                                      	     ;
stPrcRecipe.stUCF.lrCapSorterCapHightShow.lrValue			                                      	:=      stPrcRecipe.stUCF.lrCapSorterCapHightShow.lrDefault			                                      	     ;
stPrcRecipe.stUCF.lrCapSorterCapNeckHightShow.lrValue		                                      	:=      stPrcRecipe.stUCF.lrCapSorterCapNeckHightShow.lrDefault		                                      	     ;
stPrcRecipe.stUCF.lrCapSorterSpare1.lrValue                											:=      stPrcRecipe.stUCF.lrCapSorterSpare1.lrDefault	          											     ;
stPrcRecipe.stUCF.lrCapSorterSpare2.lrValue                											:=      stPrcRecipe.stUCF.lrCapSorterSpare2.lrDefault	             											 ;
stPrcRecipe.stUCF.lrCapSorterSpare3.lrValue                											:=      stPrcRecipe.stUCF.lrCapSorterSpare3.lrDefault	               											 ;
stPrcRecipe.stUCF.lrCapSorterSpare4.lrValue                											:=      stPrcRecipe.stUCF.lrCapSorterSpare4.lrDefault	            											 ;
stPrcRecipe.stUCF.lrCapSorterSpare5.lrValue                											:=      stPrcRecipe.stUCF.lrCapSorterSpare5.lrDefault	        											     ;
stPrcRecipe.stUCF.lrCapSorterSpare6.lrValue                											:=      stPrcRecipe.stUCF.lrCapSorterSpare6.lrDefault	          											     ;
stPrcRecipe.stUCF.lrCapSorterSpare7.lrValue                											:=      stPrcRecipe.stUCF.lrCapSorterSpare7.lrDefault	               											 ;
stPrcRecipe.stUBF.iBottleSorterProductTypeShow.diValue                                            	:=      stPrcRecipe.stUBF.iBottleSorterProductTypeShow.diDefault                                            	 ;
stPrcRecipe.stUBF.uiBottleSorterIndexShow.diValue		                               				:=      stPrcRecipe.stUBF.uiBottleSorterIndexShow.diDefault                             				         ;
stPrcRecipe.stUBF.bBottleSorterHopperTransporterEnableShow.bValue								  	:=      stPrcRecipe.stUBF.bBottleSorterHopperTransporterEnableShow.bDefault							  	         ;
stPrcRecipe.stUBF.iBottleSorterHopperConveyorRunningSpeedSVShow.diValue							  	:=      stPrcRecipe.stUBF.iBottleSorterHopperConveyorRunningSpeedSVShow.diDefault						  	     ;
stPrcRecipe.stUBF.iBottleSorterHopperConveyorEmptyingSpeedSVShow.diValue							:=      stPrcRecipe.stUBF.iBottleSorterHopperConveyorEmptyingSpeedSVShow.diDefault					             ;
stPrcRecipe.stUBF.iBottleSorterDistanceToFindElementOnTransferConveyorLimitRunningSVShow.diValue	:=      stPrcRecipe.stUBF.iBottleSorterDistanceToFindElementOnTransferConveyorLimitRunningSVShow.diDefault       ;
stPrcRecipe.stUBF.iBottleSorterDistanceToFindElementOnTransferConveyorLimitEmptyingSVShow.diValue 	:=      stPrcRecipe.stUBF.iBottleSorterDistanceToFindElementOnTransferConveyorLimitEmptyingSVShow.diDefault      ;
stPrcRecipe.stUBF.bBottleSorterTransferTransporterEnableShow.bValue								  	:=      stPrcRecipe.stUBF.bBottleSorterTransferTransporterEnableShow.bDefault							  	     ;
stPrcRecipe.stUBF.iBottleSorterTransferConveyorRunningSpeedSVShow.diValue						  	:=      stPrcRecipe.stUBF.iBottleSorterTransferConveyorRunningSpeedSVShow.diDefault				  	             ;
stPrcRecipe.stUBF.iBottleSorterTransferConveyorEmptyingSpeedSVShow.diValue						  	:=      stPrcRecipe.stUBF.iBottleSorterTransferConveyorEmptyingSpeedSVShow.diDefault			  	             ;
stPrcRecipe.stUBF.iBottleSorterDistanceToFindElementOnSupplyConveyorDownstairsLimitSVShow.diValue 	:=      stPrcRecipe.stUBF.iBottleSorterDistanceToFindElementOnSupplyConveyorDownstairsLimitSVShow.diDefault      ;
stPrcRecipe.stUBF.bBottleSorterSupplyTransporterEnableShow.bValue			                      	:=      stPrcRecipe.stUBF.bBottleSorterSupplyTransporterEnableShow.bDefault	                      	             ;
stPrcRecipe.stUBF.uiBottleSorterSupplyTransporterRunningSpeedSVShow.udiValue                      	:=      stPrcRecipe.stUBF.uiBottleSorterSupplyTransporterRunningSpeedSVShow.udiDefault               	         ;
stPrcRecipe.stUBF.uiBottleSorterSupplyTransporterEmptingSpeedSVShow.udiValue                      	:=      stPrcRecipe.stUBF.uiBottleSorterSupplyTransporterEmptingSpeedSVShow.udiDefault                  	     ;
stPrcRecipe.stUBF.lrBottleSorterModuloMoveOffsetSVShow.lrValue				                      	:=      stPrcRecipe.stUBF.lrBottleSorterModuloMoveOffsetSVShow.lrDefault			                      	     ;
stPrcRecipe.stUBF.iBottleSorterSensorsCountFirstConditionSVShow.diValue	                          	:=      stPrcRecipe.stUBF.iBottleSorterSensorsCountFirstConditionSVShow.diDefault                      	         ;
stPrcRecipe.stUBF.iBottleSorterSupplyTimeFirstConditionSVShow.diValue		                      	:=      stPrcRecipe.stUBF.iBottleSorterSupplyTimeFirstConditionSVShow.diDefault	                      	         ;
stPrcRecipe.stUBF.iBottleSorterSensorsCountSecondConditionMinSVShow.diValue	                      	:=      stPrcRecipe.stUBF.iBottleSorterSensorsCountSecondConditionMinSVShow.diDefault                   	     ;
stPrcRecipe.stUBF.iBottleSorterSensorsCountSecondConditionMaxSVShow.diValue	                      	:=      stPrcRecipe.stUBF.iBottleSorterSensorsCountSecondConditionMaxSVShow.diDefault            	             ;
stPrcRecipe.stUBF.iBottleSorterSupplyTimeSecondConditionSVShow.diValue		                      	:=      stPrcRecipe.stUBF.iBottleSorterSupplyTimeSecondConditionSVShow.diDefault                      	         ;
stPrcRecipe.stUBF.iBottleSorterSensorsCountThirdConditionSVShow.diValue	                          	:=      stPrcRecipe.stUBF.iBottleSorterSensorsCountThirdConditionSVShow.diDefault                       	     ;
stPrcRecipe.stUBF.iBottleSorterSupplyTimeThirdConditionSVShow.diValue		                      	:=      stPrcRecipe.stUBF.iBottleSorterSupplyTimeThirdConditionSVShow.diDefault                      	         ;
stPrcRecipe.stUBF.bBottleSorterWeelEnableShow.bValue			                       				:=      stPrcRecipe.stUBF.bBottleSorterWeelEnableShow.bDefault		                       				         ;
stPrcRecipe.stUBF.lrBottleSorterWheelSpeedSVShow.lrValue			                             	:=      stPrcRecipe.stUBF.lrBottleSorterWheelSpeedSVShow.lrDefault			                             	     ;
stPrcRecipe.stUBF.lrBottleSorterWheelEmptyingSpeedSVShow.lrValue	                              	:=      stPrcRecipe.stUBF.lrBottleSorterWheelEmptyingSpeedSVShow.lrDefault	                              	     ;
stPrcRecipe.stUBF.bBottleSorterBrushEnableShow.bValue			   									:=      stPrcRecipe.stUBF.bBottleSorterBrushEnableShow.bDefault		   									         ;
stPrcRecipe.stUBF.lrBottleSorterBrushHeightPositionSVShow.lrValue                                 	:=      stPrcRecipe.stUBF.lrBottleSorterBrushHeightPositionSVShow.lrDefault	                                	 ;
stPrcRecipe.stUBF.iBottleSorterBrushRunningSpeedSVShow.diValue	                                  	:=      stPrcRecipe.stUBF.iBottleSorterBrushRunningSpeedSVShow.diDefault                                	     ;
stPrcRecipe.stUBF.iBottleSorterBrushEmptyingSpeedSVShow.diValue	                                  	:=      stPrcRecipe.stUBF.iBottleSorterBrushEmptyingSpeedSVShow.diDefault                          	             ;
stPrcRecipe.stUBF.bBottleSorterRobotEnableShow.bValue	                            				:=      stPrcRecipe.stUBF.bBottleSorterRobotEnableShow.bDefault                            				         ;
stPrcRecipe.stUBF.nBottleSorterRobotRecipeId.udiValue		                                		:=      stPrcRecipe.stUBF.nBottleSorterRobotRecipeId.udiDefault                                		             ;
stPrcRecipe.stUBF.lrBottleSorterRemainingTimeToSuctionShow.lrValue                                	:=      stPrcRecipe.stUBF.lrBottleSorterRemainingTimeToSuctionShow.lrDefault	                                 ;
stPrcRecipe.stUBF.lrBottleSorterSuckerSuctionTimeShow.lrValue		                              	:=      stPrcRecipe.stUBF.lrBottleSorterSuckerSuctionTimeShow.lrDefault		                              	     ;
stPrcRecipe.stUBF.lrBottleSorterRemainingTimeToRejectShow.lrValue                                 	:=      stPrcRecipe.stUBF.lrBottleSorterRemainingTimeToRejectShow.lrDefault	                              	     ;
stPrcRecipe.stUBF.lrBottleSorterEjectorPulseShow.lrValue                                        	:=      stPrcRecipe.stUBF.lrBottleSorterEjectorPulseShow.lrDefault	                                      	     ;
stPrcRecipe.stUBF.lrBottleSorterZPickAboveTheBottleSVShow.lrValue	                              	:=      stPrcRecipe.stUBF.lrBottleSorterZPickAboveTheBottleSVShow.lrDefault	                             	     ;
stPrcRecipe.stUBF.lrBottleSorterZPickMoveSVShow.lrValue			                            		:=      stPrcRecipe.stUBF.lrBottleSorterZPickMoveSVShow.lrDefault			                            		 ;
stPrcRecipe.stUBF.lrBottleSorterSafetyHeightSVShow.lrValue		                              		:=      stPrcRecipe.stUBF.lrBottleSorterSafetyHeightSVShow.lrDefault		                              		 ;
stPrcRecipe.stUBF.bBottleSorterRecieverEnableShow.bValue			                              	:=      stPrcRecipe.stUBF.bBottleSorterRecieverEnableShow.bDefault		                              	         ;
stPrcRecipe.stUBF.bBottleSorterRecieverSlot1EnableShow.bValue		                              	:=      stPrcRecipe.stUBF.bBottleSorterRecieverSlot1EnableShow.bDefault                              	         ;
stPrcRecipe.stUBF.bBottleSorterRecieverSlot2EnableShow.bValue		                              	:=      stPrcRecipe.stUBF.bBottleSorterRecieverSlot2EnableShow.bDefault		                              	     ;
stPrcRecipe.stUBF.bBottleSorterRecieverSlot3EnableShow.bValue		                				:=      stPrcRecipe.stUBF.bBottleSorterRecieverSlot3EnableShow.bDefault                				             ;
stPrcRecipe.stUBF.lrBottleSorterRecieverHeightPositionSVShow.lrValue                              	:=      stPrcRecipe.stUBF.lrBottleSorterRecieverHeightPositionSVShow.lrDefault	                           	     ;
stPrcRecipe.stUCF.lrCapSorterPreScrewerPickerSpeedWhenScrewerShow.lrValue							:=		stPrcRecipe.stUCF.lrCapSorterPreScrewerPickerSpeedWhenScrewerShow.lrDefault								 ;
stPrcRecipe.stUBL.bROPPCappingEnableShow.bValue					                                    :=      stPrcRecipe.stUBL.bROPPCappingEnableShow.bDefault		                                                ;
stPrcRecipe.stUBL.bROPPDragEnableShow.bValue	 				                                    :=      stPrcRecipe.stUBL.bROPPDragEnableShow.bDefault		                                                    ;
stPrcRecipe.stUBL.bROPPFeederEnableShow.bValue					                                    :=      stPrcRecipe.stUBL.bROPPFeederEnableShow.bDefault		                                                ;
stPrcRecipe.stUBL.bROPPSlowerEnableShow.bValue	 				                                    :=      stPrcRecipe.stUBL.bROPPSlowerEnableShow.bDefault 	                                                    ;
stPrcRecipe.stUBL.iROPPCapping1ToolShow.diValue 				                                    :=      stPrcRecipe.stUBL.iROPPCapping1ToolShow.diDefault		                                                ;   
stPrcRecipe.stUBL.iROPPCappingTime2Show.diValue  				                                    :=      stPrcRecipe.stUBL.iROPPCappingTime2Show.diDefault 		                                                ;
stPrcRecipe.stUBL.iROPPCappingTimeShow.diValue  				                                    :=      stPrcRecipe.stUBL.iROPPCappingTimeShow.diDefault		                                                ;   
stPrcRecipe.stUBL.iROPPFeederTimeDelayOffShow.diValue 			                                    :=      stPrcRecipe.stUBL.iROPPFeederTimeDelayOffShow.diDefault                                                 ;
stPrcRecipe.stUBL.iROPPFeederTimeDelayOnShow.diValue  			                                    :=      stPrcRecipe.stUBL.iROPPFeederTimeDelayOnShow.diDefault                                                  ;
stPrcRecipe.stUBL.iROPPFeederTimeToEmptySleeveErrorShow.diValue	                                    :=      stPrcRecipe.stUBL.iROPPFeederTimeToEmptySleeveErrorShow.diDefault                                       ;         
stPrcRecipe.stUBL.lrROPPCappingHeightPosSVShow.lrValue			                                    :=      stPrcRecipe.stUBL.lrROPPCappingHeightPosSVShow.lrDefault	                                            ;    
stPrcRecipe.stUBL.lrROPPCappingVelocitySVShow.lrValue	 		                                    :=      stPrcRecipe.stUBL.lrROPPCappingVelocitySVShow.lrDefault	                                                ;
stPrcRecipe.stUBL.lrROPPDragAccelerationShow.lrValue	 		                                    :=      stPrcRecipe.stUBL.lrROPPDragAccelerationShow.lrDefault                                                  ;
stPrcRecipe.stUBL.lrROPPDragDecelerationShow.lrValue	 		                                    :=      stPrcRecipe.stUBL.lrROPPDragDecelerationShow.lrDefault                                                  ;
stPrcRecipe.stUBL.lrROPPDragVelocityShow.lrValue	 			                                    :=      stPrcRecipe.stUBL.lrROPPDragVelocityShow.lrDefault 	                                                    ;
stPrcRecipe.stUBL.lrROPPFeederHeightPosSVShow.lrValue	 		                                    :=      stPrcRecipe.stUBL.lrROPPFeederHeightPosSVShow.lrDefault                                  				;
stPrcRecipe.stUBL.nROPPSlowerVelocitySVShow.udiValue			                                    :=      stPrcRecipe.stUBL.nROPPSlowerVelocitySVShow.udiDefault	                                       			;
                                                                                                    
                                                                                                    
                                                                                                    
                                                                                                    
 (*                                                                                                   
                                                                                                    
stPrcRecipe.stP041_MainProcess.stProductCountX.udiValue					:=	stPrcRecipe.stP041_MainP:=rocess.stProductCountX.udiDefault;
stPrcRecipe.stP041_MainProcess.stProductCountY.udiValue					:=	stPrcRecipe.stP041_MainP:=rocess.stProductCountY.udiDefault;
stPrcRecipe.stP041_MainProcess.stProductCountZ.udiValue					:=	stPrcRecipe.stP041_MainP:=rocess.stProductCountZ.udiDefault;
stPrcRecipe.stP041_MainProcess.stProductHeight.lrValue					:=	stPrcRecipe.stP041_MainP:=rocess.stProductHeight.lrDefault;
stPrcRecipe.stP041_MainProcess.stProductSizeX.lrValue					:=	stPrcRecipe.stP041_MainP:=rocess.stProductSizeX.lrDefault;
stPrcRecipe.stP041_MainProcess.stProductSizeY.lrValue					:=	stPrcRecipe.stP041_MainP:=rocess.stProductSizeY.lrDefault;
stPrcRecipe.stP041_MainProcess.stBoxSizeX	  .	lrValue					:=	stPrcRecipe.stP041_MainProcess.stBoxSizeX	  .lrDefault;
stPrcRecipe.stP041_MainProcess.stBoxSizeY	  .lrValue				:=	stPrcRecipe.stP041_MainProcess.stBoxSizeY	  .lrDefault;
stPrcRecipe.stP041_MainProcess.stBoxSizeZ.lrValue					:=	stPrcRecipe.stP041_MainProcess.stBoxSizeZ.lrDefault;
stPrcRecipe.stP041_MainProcess.stUseBoxesTransporter.bValue					:=	stPrcRecipe.stP041_MainProcess.stUseBoxesTransporter.bDefault;
                                                                                                    
                                                                                                    
                                                                                                    
                                                                                                    
                                                                                                    
                                                                                                    
//stP100_MainSystem									:	ST_MainSystemRecipe;                        
                                                                                                    
//stP110_MachineBefore								:	ST_ExtMachineRecipe;                        
stPrcRecipe.stP110_MachineBefore.stUseComunication.bValue							:=	stPrcRecipe.stP110_MachineBefore.stUseComunication.bDefault;
                                                                                                    
//stP120_InTransporter								:	ST_InTransporterRecipe;                     
stPrcRecipe.stP120_InTransporter.stTransporterVelocity.udiValue			:=	stPrcRecipe.stP120_InTransporter.stTransporterVelocity.udiDefault;
stPrcRecipe.stP120_InTransporter.stInTransporterWidth.lrValue			:=	stPrcRecipe.stP120_InTransporter.stInTransporterWidth.lrDefault;
stPrcRecipe.stP120_InTransporter.stInTransporterLength.lrValue			:=	stPrcRecipe.stP120_InTransporter.stInTransporterLength.lrDefault;
                                                                                                    
//stP130_InGate										:	ST_StandartGateRecipe;                      
                                                                                                    
//stP131_InGate2										:	ST_StandartGateRecipe;                  
                                                                                                    
//stP140_DownCloser									:	ST_DownCloserRecipe;                        
stPrcRecipe.stP140_LeftRightCloserValve.stWidthOffset.lrValue			:=	stPrcRecipe.stP140_LeftRightCloserValve.stWidthOffset.lrDefault;
//stP141_RearCloser									:	ST_StandartGateRecipe;                      
                                                                                                    
//stP150_ProductRobot								:	ST_ProductRobotRecipe;                      
stPrcRecipe.stP150_ProductRobot.stPickOffsetX			.lrValue	:=	stPrcRecipe.stP150_ProductRobot.stPickOffsetX			.lrDefault;	 
stPrcRecipe.stP150_ProductRobot.stPickOffsetY			.lrValue	:=	stPrcRecipe.stP150_ProductRobot.stPickOffsetY			.lrDefault;	 
stPrcRecipe.stP150_ProductRobot.stPickOffsetZ			.lrValue	:=	stPrcRecipe.stP150_ProductRobot.stPickOffsetZ			.lrDefault;	 
stPrcRecipe.stP150_ProductRobot.stPickOffsetA			.lrValue	:=	stPrcRecipe.stP150_ProductRobot.stPickOffsetA			.lrDefault;	 
stPrcRecipe.stP150_ProductRobot.stPickOffsetB			.lrValue	:=	stPrcRecipe.stP150_ProductRobot.stPickOffsetB			.lrDefault;	 
stPrcRecipe.stP150_ProductRobot.stPickOffsetC			.lrValue	:=	stPrcRecipe.stP150_ProductRobot.stPickOffsetC			.lrDefault;	 
stPrcRecipe.stP150_ProductRobot.stPickAccelecation		.udiValue	:=	stPrcRecipe.stP150_ProductRobot.stPickAccelecation		.udiDefault;	 
stPrcRecipe.stP150_ProductRobot.stPickDecceleration		.udiValue	:=	stPrcRecipe.stP150_ProductRobot.stPickDecceleration		.udiDefault;	 
stPrcRecipe.stP150_ProductRobot.stPickOverride			.udiValue	:=	stPrcRecipe.stP150_ProductRobot.stPickOverride			.udiDefault;	 
stPrcRecipe.stP150_ProductRobot.stPickColisionDetect	.udiValue	:=	stPrcRecipe.stP150_ProductRobot.stPickColisionDetect	.udiDefault;	 
stPrcRecipe.stP150_ProductRobot.stPickGripperDelayTime	.udiValue	:=	stPrcRecipe.stP150_ProductRobot.stPickGripperDelayTime	.udiDefault;	 
stPrcRecipe.stP150_ProductRobot.stSuckingTimeOn		.udiValue		:=	stPrcRecipe.stP150_ProductRobot.stSuckingTimeOn		.udiDefault;	 
stPrcRecipe.stP150_ProductRobot.stSuckingTimeOff	.udiValue		:=	stPrcRecipe.stP150_ProductRobot.stSuckingTimeOff	.udiDefault;	 
stPrcRecipe.stP150_ProductRobot.stPlaceOffsetX			.lrValue	:=	stPrcRecipe.stP150_ProductRobot.stPlaceOffsetX			.lrDefault;	
stPrcRecipe.stP150_ProductRobot.stPlaceOffsetY			.lrValue	:=	stPrcRecipe.stP150_ProductRobot.stPlaceOffsetY			.lrDefault;	
stPrcRecipe.stP150_ProductRobot.stPlaceOffsetZ			.lrValue	:=	stPrcRecipe.stP150_ProductRobot.stPlaceOffsetZ			.lrDefault;	
stPrcRecipe.stP150_ProductRobot.stPlaceOffsetA			.lrValue	:=	stPrcRecipe.stP150_ProductRobot.stPlaceOffsetA			.lrDefault;	                                                                
stPrcRecipe.stP150_ProductRobot.stPlaceOffsetB			.lrValue	:=	stPrcRecipe.stP150_ProductRobot.stPlaceOffsetB			.lrDefault;	
stPrcRecipe.stP150_ProductRobot.stPlaceOffsetC			.lrValue	:=	stPrcRecipe.stP150_ProductRobot.stPlaceOffsetC			.lrDefault;	
stPrcRecipe.stP150_ProductRobot.stPlaceAccelecation		.udiValue	:=	stPrcRecipe.stP150_ProductRobot.stPlaceAccelecation		.udiDefault;	 
stPrcRecipe.stP150_ProductRobot.stPlaceDecceleration	.udiValue	:=	stPrcRecipe.stP150_ProductRobot.stPlaceDecceleration	.udiDefault;	 
stPrcRecipe.stP150_ProductRobot.stPlaceOverride			.udiValue	:=	stPrcRecipe.stP150_ProductRobot.stPlaceOverride			.udiDefault;	 
stPrcRecipe.stP150_ProductRobot.stPlaceColisionDetect	.udiValue	:=	stPrcRecipe.stP150_ProductRobot.stPlaceColisionDetect	.udiDefault;	 
stPrcRecipe.stP150_ProductRobot.stRezerwa3	.udiValue				:=	stPrcRecipe.stP150_ProductRobot.stRezerwa3	.udiDefault;	 
stPrcRecipe.stP150_ProductRobot.stRezerwa1	.udiValue				:=	stPrcRecipe.stP150_ProductRobot.stRezerwa1	.udiDefault;	 
stPrcRecipe.stP150_ProductRobot.stRezerwa2	.udiValue				:=	stPrcRecipe.stP150_ProductRobot.stRezerwa2	.udiDefault;	 
stPrcRecipe.stP150_ProductRobot.stDistanceTCP_X			.lrValue	:=	stPrcRecipe.stP150_ProductRobot.stDistanceTCP_X			.lrDefault;	 
stPrcRecipe.stP150_ProductRobot.stDistanceTCP_Y			.lrValue	:=	stPrcRecipe.stP150_ProductRobot.stDistanceTCP_Y			.lrDefault;	 
stPrcRecipe.stP150_ProductRobot.stDistanceTCP_Z			.lrValue	:=	stPrcRecipe.stP150_ProductRobot.stDistanceTCP_Z			.lrDefault;	 
stPrcRecipe.stP150_ProductRobot.stPickPreX				.lrValue	:=	stPrcRecipe.stP150_ProductRobot.stPickPreX				.lrDefault;	 
stPrcRecipe.stP150_ProductRobot.stPickPreY				.lrValue	:=	stPrcRecipe.stP150_ProductRobot.stPickPreY				.lrDefault;	 
stPrcRecipe.stP150_ProductRobot.stPickPreZ				.lrValue	:=	stPrcRecipe.stP150_ProductRobot.stPickPreZ				.lrDefault;	 
stPrcRecipe.stP150_ProductRobot.stPickAfterX			.lrValue	:=	stPrcRecipe.stP150_ProductRobot.stPickAfterX			.lrDefault;	 
stPrcRecipe.stP150_ProductRobot.stPickAfterY		    .lrValue	:=	stPrcRecipe.stP150_ProductRobot.stPickAfterY		    .lrDefault;	 
stPrcRecipe.stP150_ProductRobot.stPickAfterZ		    .lrValue	:=	stPrcRecipe.stP150_ProductRobot.stPickAfterZ		    .lrDefault;		
stPrcRecipe.stP150_ProductRobot.stAfterPickSafeX		.lrValue	:=	stPrcRecipe.stP150_ProductRobot.stAfterPickSafeX		.lrDefault;	 
stPrcRecipe.stP150_ProductRobot.stPlacePreX				.lrValue	:=	stPrcRecipe.stP150_ProductRobot.stPlacePreX				.lrDefault;	 
stPrcRecipe.stP150_ProductRobot.stPlacePreY		        .lrValue	:=	stPrcRecipe.stP150_ProductRobot.stPlacePreY		        .lrDefault;	 
stPrcRecipe.stP150_ProductRobot.stPlacePreZ		        .lrValue	:=	stPrcRecipe.stP150_ProductRobot.stPlacePreZ		        .lrDefault;	 
stPrcRecipe.stP150_ProductRobot.stPlaceAfterX		    .lrValue	:=	stPrcRecipe.stP150_ProductRobot.stPlaceAfterX		    .lrDefault;	 
stPrcRecipe.stP150_ProductRobot.stPlaceAfterY		    .lrValue	:=	stPrcRecipe.stP150_ProductRobot.stPlaceAfterY		    .lrDefault;	 
stPrcRecipe.stP150_ProductRobot.stPlaceAfterZ		    .lrValue	:=	stPrcRecipe.stP150_ProductRobot.stPlaceAfterZ		    .lrDefault;	 
stPrcRecipe.stP150_ProductRobot.stProductHighOffsetZ	.lrValue	:=	stPrcRecipe.stP150_ProductRobot.stProductHighOffsetZ	        .lrDefault;	 
stPrcRecipe.stP150_ProductRobot.stProductPickHeight		.lrValue	:=	stPrcRecipe.stP150_ProductRobot.stProductPickHeight		.lrDefault;


//stP151_GateBeforeRobot							:	ST_StandartGateRecipe;
							
//stP160_MoverStepMotor								:	ST_StepMoverRecipe;
stPrcRecipe.stP160_MoverStepMotor.stLowAcceleration.lrValue							:=	stPrcRecipe.stP160_MoverStepMotor.stLowAcceleration.lrDefault;
stPrcRecipe.stP160_MoverStepMotor.stLowDeceleration.lrValue							:=	stPrcRecipe.stP160_MoverStepMotor.stLowDeceleration.lrDefault;
stPrcRecipe.stP160_MoverStepMotor.stLowJerk.lrValue									:=	stPrcRecipe.stP160_MoverStepMotor.stLowJerk.lrDefault;
stPrcRecipe.stP160_MoverStepMotor.stLowVelocity.lrValue								:=	stPrcRecipe.stP160_MoverStepMotor.stLowVelocity.lrDefault;

stPrcRecipe.stP160_MoverStepMotor.stHighAcceleration.lrValue							:=	stPrcRecipe.stP160_MoverStepMotor.stHighAcceleration.lrDefault;
stPrcRecipe.stP160_MoverStepMotor.stHighDeceleration.lrValue							:=	stPrcRecipe.stP160_MoverStepMotor.stHighDeceleration.lrDefault;
stPrcRecipe.stP160_MoverStepMotor.stHighJerk.lrValue									:=	stPrcRecipe.stP160_MoverStepMotor.stHighJerk.lrDefault;
stPrcRecipe.stP160_MoverStepMotor.stHighVelocity.lrValue								:=	stPrcRecipe.stP160_MoverStepMotor.stHighVelocity.lrDefault;

//stP161_MoverPneumo1								:	ST_StandartGateRecipe;

//stP162_MoverPneumo2Long							:	ST_StandartGateRecipe;

//stP163_MoverPneumo2Short							:	ST_StandartGateRecipe;

//stP164_MoverVacuum1								:	ST_SucterRecipe;

//stP165_MoverVacuum2								:	ST_SucterRecipe;

//stP170_CornerSupport								:	ST_StandartGateRecipe;

//stP180_LiftedTable								:	ST_LiftedTableRecipe;

//stP190_BoxFeeder									:	ST_BoxFeederRecipe;


//stP200_BoxRobot									:	ST_BoxRobotRecipe;
stPrcRecipe.stP200_BoxRobot.stPickOffsetX			.lrValue				:=	stPrcRecipe.stP200_BoxRobot.stPickOffsetX			.lrDefault;	
stPrcRecipe.stP200_BoxRobot.stPickOffsetY			.lrValue				:=	stPrcRecipe.stP200_BoxRobot.stPickOffsetY			.lrDefault;	
stPrcRecipe.stP200_BoxRobot.stPickOffsetZ			.lrValue				:=	stPrcRecipe.stP200_BoxRobot.stPickOffsetZ			.lrDefault;	
stPrcRecipe.stP200_BoxRobot.stPickOffsetA			.lrValue				:=	stPrcRecipe.stP200_BoxRobot.stPickOffsetA			.lrDefault;	
stPrcRecipe.stP200_BoxRobot.stPickOffsetB			.lrValue				:=	stPrcRecipe.stP200_BoxRobot.stPickOffsetB			.lrDefault;	
stPrcRecipe.stP200_BoxRobot.stPickOffsetC			.lrValue				:=	stPrcRecipe.stP200_BoxRobot.stPickOffsetC			.lrDefault;	
                                                                                
stPrcRecipe.stP200_BoxRobot.stPickAccelecation		.udiValue				:=	stPrcRecipe.stP200_BoxRobot.stPickAccelecation		.udiDefault;	
stPrcRecipe.stP200_BoxRobot.stPickDecceleration		.udiValue				:=	stPrcRecipe.stP200_BoxRobot.stPickDecceleration		.udiDefault;	
stPrcRecipe.stP200_BoxRobot.stPickOverride			.udiValue				:=	stPrcRecipe.stP200_BoxRobot.stPickOverride			.udiDefault;	
stPrcRecipe.stP200_BoxRobot.stPickColisionDetect	.udiValue				:=	stPrcRecipe.stP200_BoxRobot.stPickColisionDetect	.udiDefault;	
stPrcRecipe.stP200_BoxRobot.stPickGripperDelayTime	.udiValue				:=	stPrcRecipe.stP200_BoxRobot.stPickGripperDelayTime	.udiDefault;	
stPrcRecipe.stP200_BoxRobot.stSuckingTimeOn		.udiValue				:=	stPrcRecipe.stP200_BoxRobot.stSuckingTimeOn		.udiDefault;	
stPrcRecipe.stP200_BoxRobot.stSuckingTimeOff	.udiValue				:=	stPrcRecipe.stP200_BoxRobot.stSuckingTimeOff	.udiDefault;	
                                                                                
stPrcRecipe.stP200_BoxRobot.stPlaceOffsetX			.lrValue				:=	stPrcRecipe.stP200_BoxRobot.stPlaceOffsetX			.lrDefault;	
stPrcRecipe.stP200_BoxRobot.stPlaceOffsetY			.lrValue				:=	stPrcRecipe.stP200_BoxRobot.stPlaceOffsetY			.lrDefault;	
stPrcRecipe.stP200_BoxRobot.stPlaceOffsetZ			.lrValue				:=	stPrcRecipe.stP200_BoxRobot.stPlaceOffsetZ			.lrDefault;	
stPrcRecipe.stP200_BoxRobot.stPlaceOffsetA			.lrValue    			:=	stPrcRecipe.stP200_BoxRobot.stPlaceOffsetA			.lrDefault;    
stPrcRecipe.stP200_BoxRobot.stPlaceOffsetB			.lrValue    			:=	stPrcRecipe.stP200_BoxRobot.stPlaceOffsetB			.lrDefault;    
stPrcRecipe.stP200_BoxRobot.stPlaceOffsetC			.lrValue                :=  stPrcRecipe.stP200_BoxRobot.stPlaceOffsetC			.lrDefault;    
                                                                                
stPrcRecipe.stP200_BoxRobot.stPlaceAccelecation		.udiValue   	        :=  stPrcRecipe.stP200_BoxRobot.stPlaceAccelecation		.udiDefault;   
stPrcRecipe.stP200_BoxRobot.stPlaceDecceleration	.udiValue   	        :=  stPrcRecipe.stP200_BoxRobot.stPlaceDecceleration	.udiDefault;   
stPrcRecipe.stP200_BoxRobot.stPlaceOverride			.udiValue   	        :=  stPrcRecipe.stP200_BoxRobot.stPlaceOverride			.udiDefault;   
stPrcRecipe.stP200_BoxRobot.stPlaceColisionDetect	.udiValue   	        :=  stPrcRecipe.stP200_BoxRobot.stPlaceColisionDetect	.udiDefault;   
stPrcRecipe.stP200_BoxRobot.stRezerwa3	.udiValue               :=  stPrcRecipe.stP200_BoxRobot.stRezerwa3	.udiDefault;   
stPrcRecipe.stP200_BoxRobot.stRezerwa1	.udiValue   	        :=  stPrcRecipe.stP200_BoxRobot.stRezerwa1	.udiDefault;   
stPrcRecipe.stP200_BoxRobot.stRezerwa2	.udiValue   	        :=  stPrcRecipe.stP200_BoxRobot.stRezerwa2	.udiDefault;   
stPrcRecipe.stP200_BoxRobot.stGripperTimeOpen		.udiValue   	        :=  stPrcRecipe.stP200_BoxRobot.stGripperTimeOpen		.udiDefault;   
stPrcRecipe.stP200_BoxRobot.stGripperTimeClose		.udiValue   	        :=  stPrcRecipe.stP200_BoxRobot.stGripperTimeClose		.udiDefault;   
                                                                              
stPrcRecipe.stP200_BoxRobot.stPickPreX				.lrValue    	        :=  stPrcRecipe.stP200_BoxRobot.stPickPreX				.lrDefault;    
stPrcRecipe.stP200_BoxRobot.stPickPreY				.lrValue    	        :=  stPrcRecipe.stP200_BoxRobot.stPickPreY				.lrDefault;    
stPrcRecipe.stP200_BoxRobot.stPickPreZ				.lrValue    	        :=  stPrcRecipe.stP200_BoxRobot.stPickPreZ				.lrDefault;    
stPrcRecipe.stP200_BoxRobot.stPickAfterX			.lrValue    	        :=  stPrcRecipe.stP200_BoxRobot.stPickAfterX			.lrDefault;    
stPrcRecipe.stP200_BoxRobot.stPickAfterY		    .lrValue    	        :=  stPrcRecipe.stP200_BoxRobot.stPickAfterY		    .lrDefault;    
stPrcRecipe.stP200_BoxRobot.stPickAfterZ		    .lrValue    	        :=  stPrcRecipe.stP200_BoxRobot.stPickAfterZ		    .lrDefault;    
stPrcRecipe.stP200_BoxRobot.stPlacePreX				.lrValue		        :=  stPrcRecipe.stP200_BoxRobot.stPlacePreX				.lrDefault;	
stPrcRecipe.stP200_BoxRobot.stPlacePreY		        .lrValue    	        :=  stPrcRecipe.stP200_BoxRobot.stPlacePreY		        .lrDefault;    
stPrcRecipe.stP200_BoxRobot.stPlacePreZ		        .lrValue    	        :=  stPrcRecipe.stP200_BoxRobot.stPlacePreZ		        .lrDefault;    
stPrcRecipe.stP200_BoxRobot.stPlaceAfterX		    .lrValue    	        :=  stPrcRecipe.stP200_BoxRobot.stPlaceAfterX		    .lrDefault;    
stPrcRecipe.stP200_BoxRobot.stPlaceAfterY		    .lrValue    	        :=  stPrcRecipe.stP200_BoxRobot.stPlaceAfterY		    .lrDefault;    
stPrcRecipe.stP200_BoxRobot.stPlaceAfterZ		    .lrValue    	        :=  stPrcRecipe.stP200_BoxRobot.stPlaceAfterZ		    .lrDefault;    
stPrcRecipe.stP200_BoxRobot.stBoxPickHeight			.lrValue				:=	stPrcRecipe.stP200_BoxRobot.stBoxPickHeight.lrDefault;
stPrcRecipe.stP200_BoxRobot.stBoxWingDown	  	    .lrValue    	        :=  stPrcRecipe.stP200_BoxRobot.stBoxWingDown	  	    .lrDefault;    
stPrcRecipe.stP200_BoxRobot.stCurveMotionPositionZ	  	    .lrValue    	        :=  stPrcRecipe.stP200_BoxRobot.stCurveMotionPositionZ	  	    .lrDefault;    
stPrcRecipe.stP200_BoxRobot.stCurveDistanceX	    .lrValue    	        :=  stPrcRecipe.stP200_BoxRobot.stCurveDistanceX	    .lrDefault;    
stPrcRecipe.stP200_BoxRobot.stCurveDistanceY		.lrValue    	        :=  stPrcRecipe.stP200_BoxRobot.stCurveDistanceY		.lrDefault;    
stPrcRecipe.stP200_BoxRobot.stCurveDistanceZ	    .lrValue    	        :=  stPrcRecipe.stP200_BoxRobot.stCurveDistanceZ	    .lrDefault;    
stPrcRecipe.stP200_BoxRobot.stCurveMotionAngleA		.lrValue		        :=  stPrcRecipe.stP200_BoxRobot.stCurveMotionAngleA		.lrDefault;	
stPrcRecipe.stP200_BoxRobot.stCurveMotionAngleB     .lrValue		        :=  stPrcRecipe.stP200_BoxRobot.stCurveMotionAngleB     .lrDefault;	

//stP230_OutControl									:	ST_OutControlRecipe;
stPrcRecipe.stP230_OutControl.stUseControl.bValue									:=	stPrcRecipe.stP230_OutControl.stUseControl.bDefault;
stPrcRecipe.stP230_OutControl.stMaxWaitSensorTime.udiValue							:=	stPrcRecipe.stP230_OutControl.stMaxWaitSensorTime.udiDefault;

//stP240_MachineNext								:	ST_ExtMachineRecipe;
stPrcRecipe.stP240_MachineNext.stUseComunication.bValue								:=	stPrcRecipe.stP240_MachineNext.stUseComunication.bDefault;

